// Mitsubishi GX Works2 project: Conv_TF_Connect_Kanban   PLC: FX3U/FX3UC

// global labels: Proce_C1
VAR_GLOBAL
  Add_Plates_C1 : INT;
  Pre_Add_Plates_C1 : INT;
  Add_Box_C1 : INT;
  Out_Product_C1 : INT;
  Codition_C2 : BOOL;
END_VAR

// global labels: Fake_Data
VAR_GLOBAL
  Fake_M45 : TIMER;
END_VAR

PROGRAM ARLAM
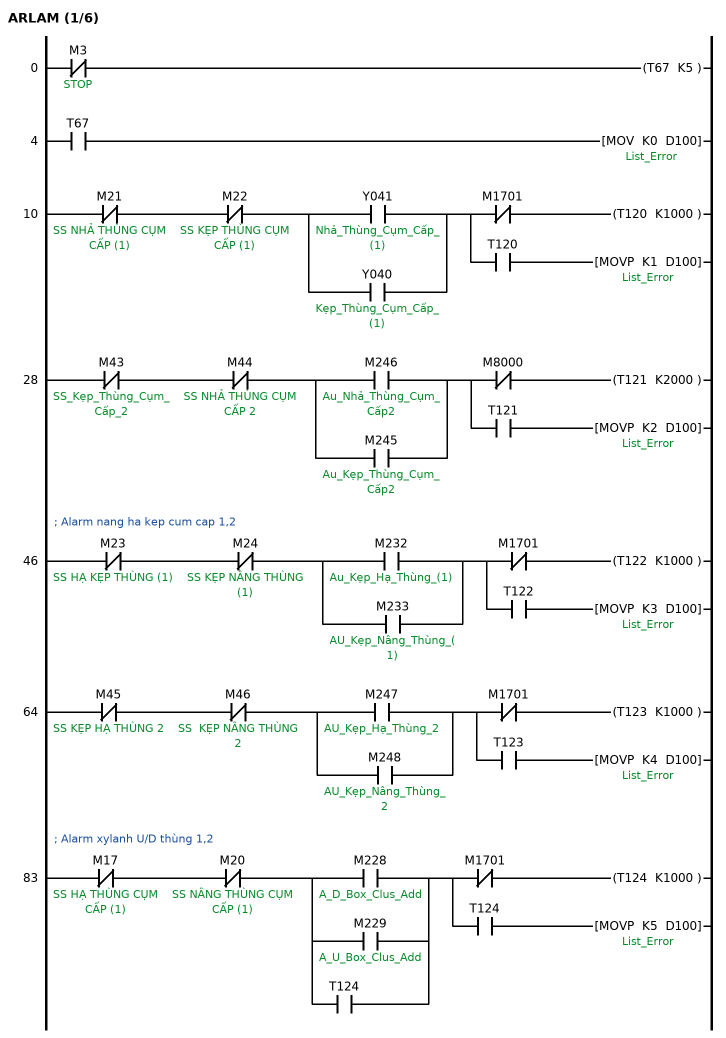
0     LDI     M3  ; STOP
      OUT     T67 K5
4     LD      T67
      MOV     K0 D100  ; List_Error
10    LDI     M21  ; SS NHẢ THÙNG CỤM CẤP (1)
      ANI     M22  ; SS KẸP THÙNG CỤM CẤP (1)
      LD      Y041  ; Nhả_Thùng_Cụm_Cấp_(1)
      OR      Y040  ; Kẹp_Thùng_Cụm_Cấp_(1)
      ANB
      MPS
      ANI     M1701
      OUT     T120 K1000
      MPP
      AND     T120
      MOVP    K1 D100
28    LDI     M43  ; SS_Kẹp_Thùng_Cụm_Cấp_2
      ANI     M44  ; SS NHẢ THÙNG CỤM CẤP 2
      LD      M246  ; Au_Nhả_Thùng_Cụm_Cấp2
      OR      M245  ; Au_Kẹp_Thùng_Cụm_Cấp2
      ANB
      MPS
      ANI     M8000
      OUT     T121 K2000
      MPP
      AND     T121
      MOVP    K2 D100
; Alarm nang ha kep cum cap 1,2
46    LDI     M23  ; SS HẠ KẸP THÙNG (1)
      ANI     M24  ; SS KẸP NÂNG THÙNG (1)
      LD      M232  ; Au_Kẹp_Hạ_Thùng_(1)
      OR      M233  ; AU_Kẹp_Nâng_Thùng_(1)
      ANB
      MPS
      ANI     M1701
      OUT     T122 K1000
      MPP
      AND     T122
      MOVP    K3 D100
64    LDI     M45  ; SS KẸP HẠ THÙNG 2
      ANI     M46  ; SS  KẸP NÂNG THÙNG 2
      LD      M247  ; AU_Kẹp_Hạ_Thùng_2
      OR      M248  ; AU_Kẹp_Nâng_Thùng_2
      ANB
      MPS
      ANI     M1701
      OUT     T123 K1000
      MPP
      AND     T123
      MOVP    K4 D100
; Alarm xylanh U/D thùng 1,2
83    LDI     M17  ; SS HẠ THÙNG CỤM CẤP (1)
      ANI     M20  ; SS NÂNG THÙNG CỤM CẤP (1)
      LD      M228  ; A_D_Box_Clus_Add
      OR      M229  ; A_U_Box_Clus_Add
      OR      T124
      ANB
      MPS
      ANI     M1701
      OUT     T124 K1000
      MPP
      AND     T124
      MOVP    K5 D100
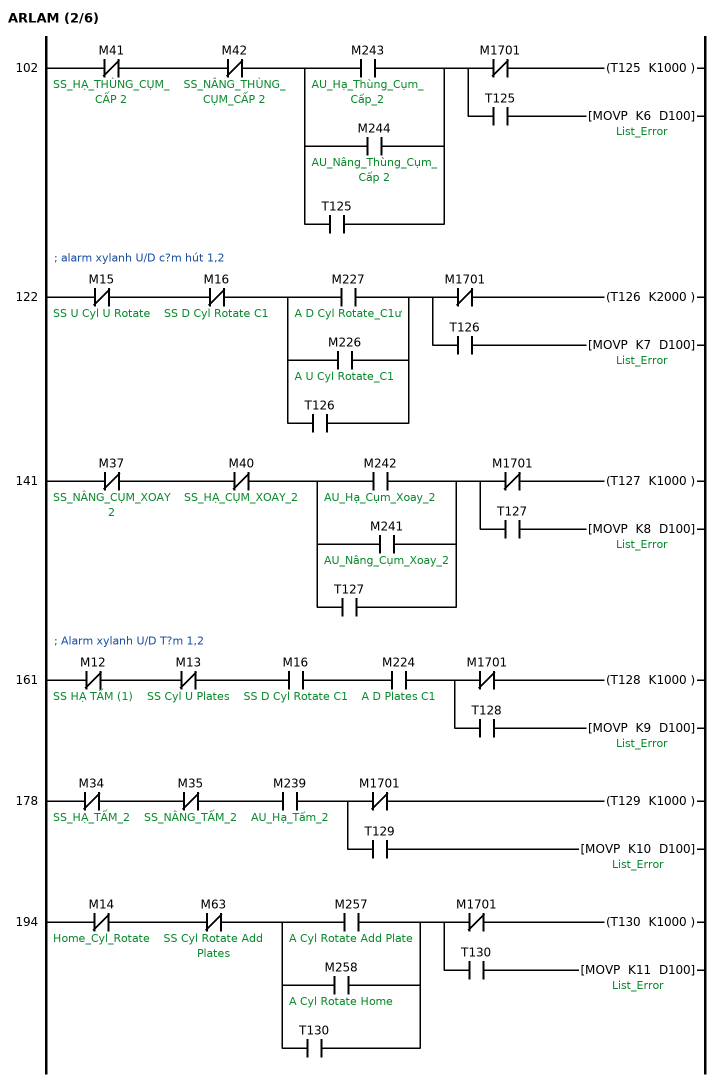
102   LDI     M41  ; SS_HẠ_THÙNG_CỤM_CẤP 2
      ANI     M42  ; SS_NÂNG_THÙNG_CỤM_CẤP 2
      LD      M243  ; AU_Hạ_Thùng_Cụm_Cấp_2
      OR      M244  ; AU_Nâng_Thùng_Cụm_Cấp 2
      OR      T125
      ANB
      MPS
      ANI     M1701
      OUT     T125 K1000
      MPP
      AND     T125
      MOVP    K6 D100
; alarm xylanh U/D c?m hút 1,2
122   LDI     M15  ; SS U Cyl U Rotate
      ANI     M16  ; SS D Cyl Rotate C1
      LD      M227  ; A D Cyl Rotate_C1ư
      OR      M226  ; A U Cyl Rotate_C1
      OR      T126
      ANB
      MPS
      ANI     M1701
      OUT     T126 K2000
      MPP
      AND     T126
      MOVP    K7 D100
141   LDI     M37  ; SS_NÂNG_CỤM_XOAY 2
      ANI     M40  ; SS_HẠ_CỤM_XOAY_2
      LD      M242  ; AU_Hạ_Cụm_Xoay_2
      OR      M241  ; AU_Nâng_Cụm_Xoay_2
      OR      T127
      ANB
      MPS
      ANI     M1701
      OUT     T127 K1000
      MPP
      AND     T127
      MOVP    K8 D100
; Alarm xylanh U/D T?m 1,2
161   LDI     M12  ; SS HẠ TẤM (1)
      ANI     M13  ; SS Cyl U Plates
      AND     M16  ; SS D Cyl Rotate C1
      AND     M224  ; A D Plates C1
      MPS
      ANI     M1701
      OUT     T128 K1000
      MPP
      AND     T128
      MOVP    K9 D100
178   LDI     M34  ; SS_HẠ_TẤM_2
      ANI     M35  ; SS_NÂNG_TẤM_2
      AND     M239  ; AU_Hạ_Tấm_2
      MPS
      ANI     M1701
      OUT     T129 K1000
      MPP
      AND     T129
      MOVP    K10 D100
194   LDI     M14  ; Home_Cyl_Rotate
      ANI     M63  ; SS Cyl Rotate Add Plates
      LD      M257  ; A Cyl Rotate Add Plate
      OR      M258  ; A Cyl Rotate Home
      OR      T130
      ANB
      MPS
      ANI     M1701
      OUT     T130 K1000
      MPP
      AND     T130
      MOVP    K11 D100
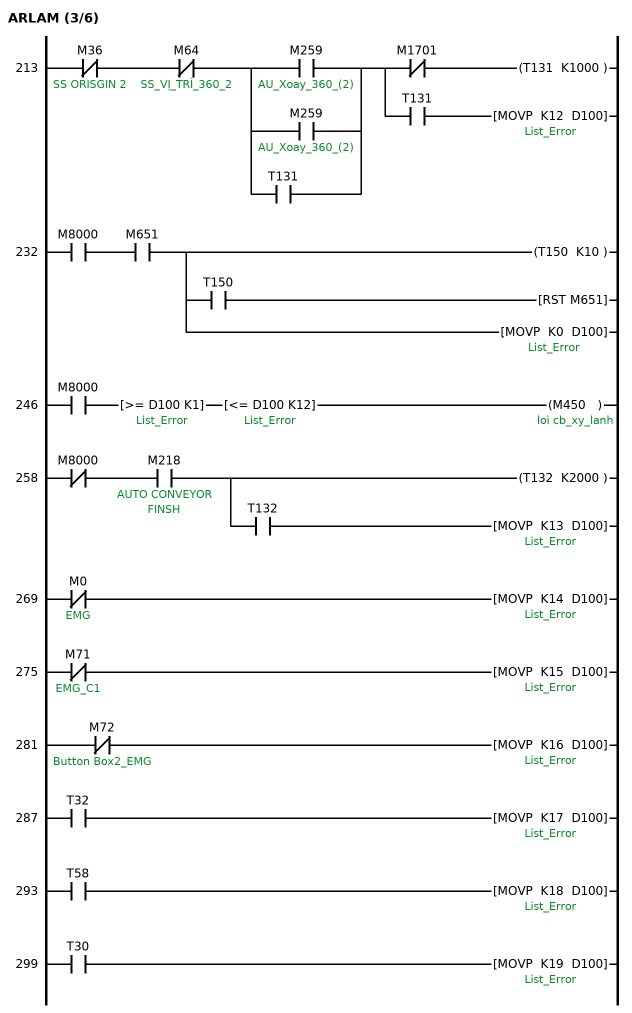
213   LDI     M36  ; SS ORISGIN 2
      ANI     M64  ; SS_VỊ_TRÍ_360_2
      LD      M259  ; AU_Xoay_360_(2)
      OR      M259  ; AU_Xoay_360_(2)
      OR      T131
      ANB
      MPS
      ANI     M1701
      OUT     T131 K1000
      MPP
      AND     T131
      MOVP    K12 D100
232   LD      M8000
      AND     M651
      OUT     T150 K10
      MPS
      AND     T150
      RST     M651
      MPP
      MOVP    K0 D100
246   LD      M8000
      AND>=   D100 K1  ; List_Error
      AND<=   D100 K12  ; List_Error
      OUT     M450  ; loi cb_xy_lanh
258   LDI     M8000
      AND     M218  ; AUTO CONVEYOR FINSH
      OUT     T132 K2000
      AND     T132
      MOVP    K13 D100
269   LDI     M0  ; EMG
      MOVP    K14 D100
275   LDI     M71  ; EMG_C1
      MOVP    K15 D100
281   LDI     M72  ; Button Box2_EMG
      MOVP    K16 D100
287   LD      T32
      MOVP    K17 D100
293   LD      T58
      MOVP    K18 D100
299   LD      T30
      MOVP    K19 D100
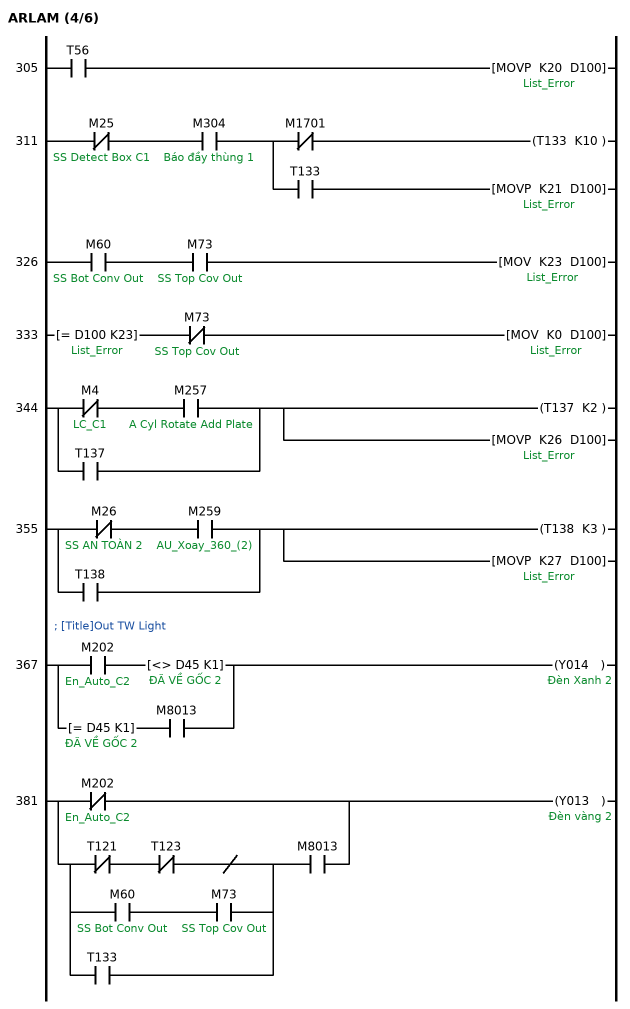
305   LD      T56
      MOVP    K20 D100
311   LDI     M25  ; SS Detect Box C1
      AND     M304  ; Báo đầy thùng 1
      MPS
      ANI     M1701
      OUT     T133 K10
      MPP
      AND     T133
      MOVP    K21 D100
326   LD      M60  ; SS Bot Conv Out
      AND     M73  ; SS Top Cov Out
      MOV     K23 D100
333   LD=     D100 K23  ; List_Error
      ANI     M73  ; SS Top Cov Out
      MOV     K0 D100
344   LDI     M4  ; LC_C1
      AND     M257  ; A Cyl Rotate Add Plate
      OR      T137
      OUT     T137 K2
      MOVP    K26 D100
355   LDI     M26  ; SS AN TOÀN 2
      AND     M259  ; AU_Xoay_360_(2)
      OR      T138
      OUT     T138 K3
      MOVP    K27 D100
; [Title]Out TW Light
367   LD      M202  ; En_Auto_C2
      AND<>   D45 K1  ; ĐÃ VỀ GỐC 2
      LD=     D45 K1  ; ĐÃ VỀ GỐC 2
      AND     M8013
      ORB
      OUT     Y014  ; Đèn Xanh 2
381   LDI     M202  ; En_Auto_C2
      LDI     T121
      ANI     T123
      INV
      LD      M60  ; SS Bot Conv Out
      AND     M73  ; SS Top Cov Out
      ORB
      OR      T133
      AND     M8013
      ORB
      OUT     Y013  ; Đèn vàng 2
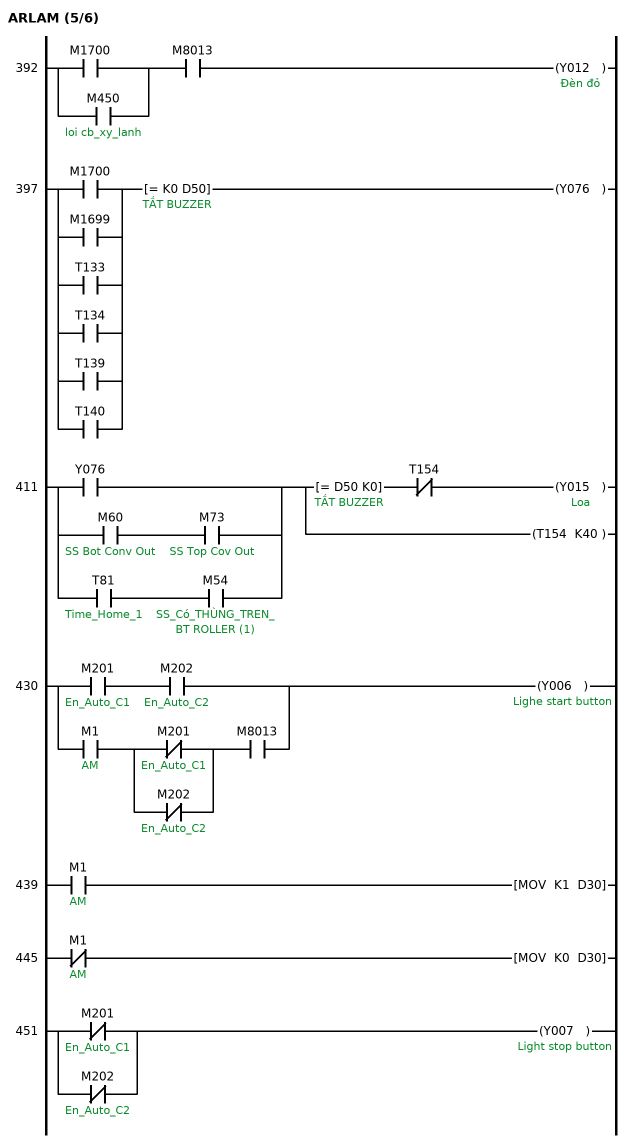
392   LD      M1700
      OR      M450  ; loi cb_xy_lanh
      AND     M8013
      OUT     Y012  ; Đèn đỏ
397   LD      M1700
      OR      M1699
      OR      T133
      OR      T134
      OR      T139
      OR      T140
      AND=    K0 D50  ; TẮT BUZZER
      OUT     Y076
411   LD      Y076
      LD      M60  ; SS Bot Conv Out
      AND     M73  ; SS Top Cov Out
      ORB
      LD      T81  ; Time_Home_1
      AND     M54  ; SS_Có_THÙNG_TREN_BT ROLLER (1)
      ORB
      MPS
      AND=    D50 K0  ; TẮT BUZZER
      ANI     T154
      OUT     Y015  ; Loa
      MPP
      OUT     T154 K40
430   LD      M201  ; En_Auto_C1
      AND     M202  ; En_Auto_C2
      LD      M1  ; AM
      LDI     M201  ; En_Auto_C1
      ORI     M202  ; En_Auto_C2
      ANB
      AND     M8013
      ORB
      OUT     Y006  ; Lighe start button
439   LD      M1  ; AM
      MOV     K1 D30
445   LDI     M1  ; AM
      MOV     K0 D30
451   LDI     M201  ; En_Auto_C1
      ORI     M202  ; En_Auto_C2
      OUT     Y007  ; Light stop button
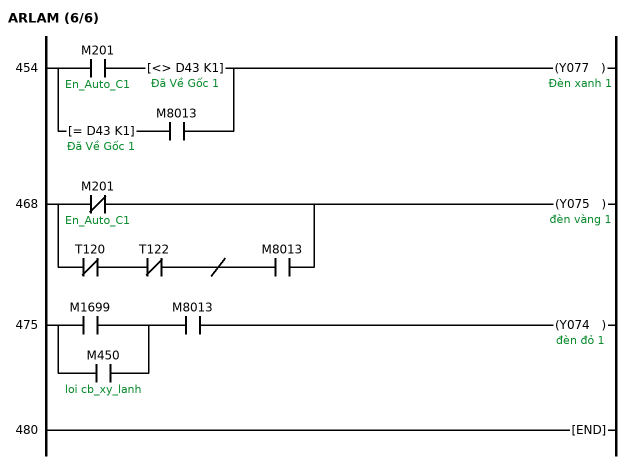
454   LD      M201  ; En_Auto_C1
      AND<>   D43 K1  ; Đã Về Gốc 1
      LD=     D43 K1  ; Đã Về Gốc 1
      AND     M8013
      ORB
      OUT     Y077  ; Đèn xanh 1
468   LDI     M201  ; En_Auto_C1
      LDI     T120
      ANI     T122
      INV
      AND     M8013
      ORB
      OUT     Y075  ; đèn vàng 1
475   LD      M1699
      OR      M450  ; loi cb_xy_lanh
      AND     M8013
      OUT     Y074  ; đèn đỏ 1
480   END
END_PROGRAM

PROGRAM AUTO
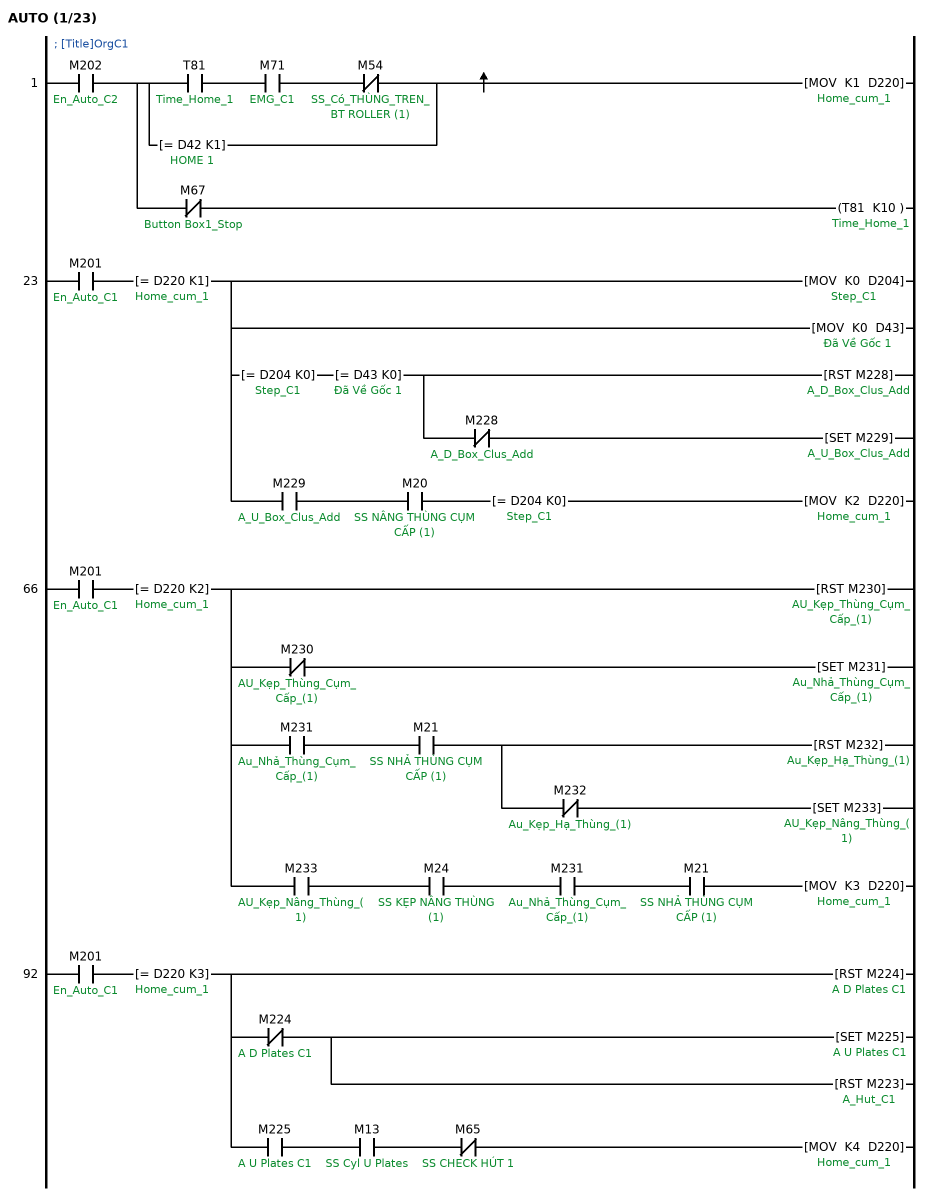
; [Title]OrgC1
1     LD      M202  ; En_Auto_C2
      MPS
      LD      T81  ; Time_Home_1
      AND     M71  ; EMG_C1
      ANI     M54  ; SS_Có_THÙNG_TREN_BT ROLLER (1)
      OR=     D42 K1  ; HOME 1
      ANB
      MEP
      MOV     K1 D220  ; Home_cum_1
      MPP
      ANI     M67  ; Button Box1_Stop
      OUT     T81 K10  ; Time_Home_1
23    LD      M201  ; En_Auto_C1
      AND=    D220 K1  ; Home_cum_1
      MOV     K0 D204  ; Step_C1
      MOV     K0 D43  ; Đã Về Gốc 1
      MPS
      AND=    D204 K0  ; Step_C1
      AND=    D43 K0  ; Đã Về Gốc 1
      RST     M228  ; A_D_Box_Clus_Add
      ANI     M228  ; A_D_Box_Clus_Add
      SET     M229  ; A_U_Box_Clus_Add
      MPP
      AND     M229  ; A_U_Box_Clus_Add
      AND     M20  ; SS NÂNG THÙNG CỤM CẤP (1)
      AND=    D204 K0  ; Step_C1
      MOV     K2 D220
66    LD      M201  ; En_Auto_C1
      AND=    D220 K2  ; Home_cum_1
      RST     M230  ; AU_Kẹp_Thùng_Cụm_Cấp_(1)
      MPS
      ANI     M230  ; AU_Kẹp_Thùng_Cụm_Cấp_(1)
      SET     M231  ; Au_Nhả_Thùng_Cụm_Cấp_(1)
      MRD
      AND     M231  ; Au_Nhả_Thùng_Cụm_Cấp_(1)
      AND     M21  ; SS NHẢ THÙNG CỤM CẤP (1)
      RST     M232  ; Au_Kẹp_Hạ_Thùng_(1)
      ANI     M232  ; Au_Kẹp_Hạ_Thùng_(1)
      SET     M233  ; AU_Kẹp_Nâng_Thùng_(1)
      MPP
      AND     M233  ; AU_Kẹp_Nâng_Thùng_(1)
      AND     M24  ; SS KẸP NÂNG THÙNG (1)
      AND     M231  ; Au_Nhả_Thùng_Cụm_Cấp_(1)
      AND     M21  ; SS NHẢ THÙNG CỤM CẤP (1)
      MOV     K3 D220
92    LD      M201  ; En_Auto_C1
      AND=    D220 K3  ; Home_cum_1
      RST     M224  ; A D Plates C1
      MPS
      ANI     M224  ; A D Plates C1
      SET     M225  ; A U Plates C1
      RST     M223  ; A_Hut_C1
      MPP
      AND     M225  ; A U Plates C1
      AND     M13  ; SS Cyl U Plates
      ANI     M65  ; SS CHECK HÚT 1
      MOV     K4 D220
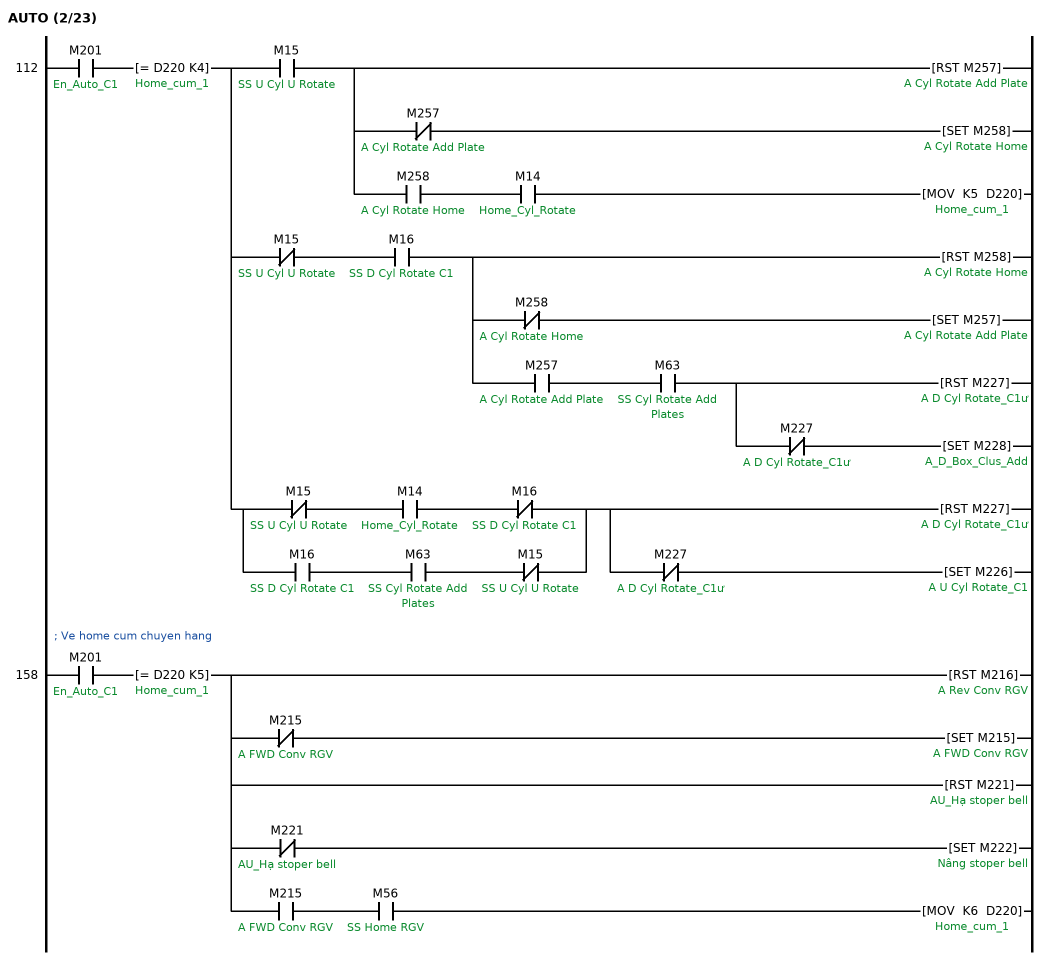
112   LD      M201  ; En_Auto_C1
      AND=    D220 K4  ; Home_cum_1
      MPS
      AND     M15  ; SS U Cyl U Rotate
      RST     M257  ; A Cyl Rotate Add Plate
      MPS
      ANI     M257  ; A Cyl Rotate Add Plate
      SET     M258  ; A Cyl Rotate Home
      MPP
      AND     M258  ; A Cyl Rotate Home
      AND     M14  ; Home_Cyl_Rotate
      MOV     K5 D220
      MRD
      ANI     M15  ; SS U Cyl U Rotate
      AND     M16  ; SS D Cyl Rotate C1
      RST     M258  ; A Cyl Rotate Home
      MPS
      ANI     M258  ; A Cyl Rotate Home
      SET     M257  ; A Cyl Rotate Add Plate
      MPP
      AND     M257  ; A Cyl Rotate Add Plate
      AND     M63  ; SS Cyl Rotate Add Plates
      RST     M227  ; A D Cyl Rotate_C1ư
      ANI     M227  ; A D Cyl Rotate_C1ư
      SET     M228  ; A_D_Box_Clus_Add
      MPP
      LDI     M15  ; SS U Cyl U Rotate
      AND     M14  ; Home_Cyl_Rotate
      ANI     M16  ; SS D Cyl Rotate C1
      LD      M16  ; SS D Cyl Rotate C1
      AND     M63  ; SS Cyl Rotate Add Plates
      ANI     M15  ; SS U Cyl U Rotate
      ORB
      ANB
      RST     M227  ; A D Cyl Rotate_C1ư
      ANI     M227  ; A D Cyl Rotate_C1ư
      SET     M226  ; A U Cyl Rotate_C1
; Ve home cum chuyen hang
158   LD      M201  ; En_Auto_C1
      AND=    D220 K5  ; Home_cum_1
      RST     M216  ; A Rev Conv RGV
      MPS
      ANI     M215  ; A FWD Conv RGV
      SET     M215  ; A FWD Conv RGV
      MPP
      RST     M221  ; AU_Hạ stoper bell
      MPS
      ANI     M221  ; AU_Hạ stoper bell
      SET     M222  ; Nâng stoper bell
      MPP
      AND     M215  ; A FWD Conv RGV
      AND     M56  ; SS Home RGV
      MOV     K6 D220
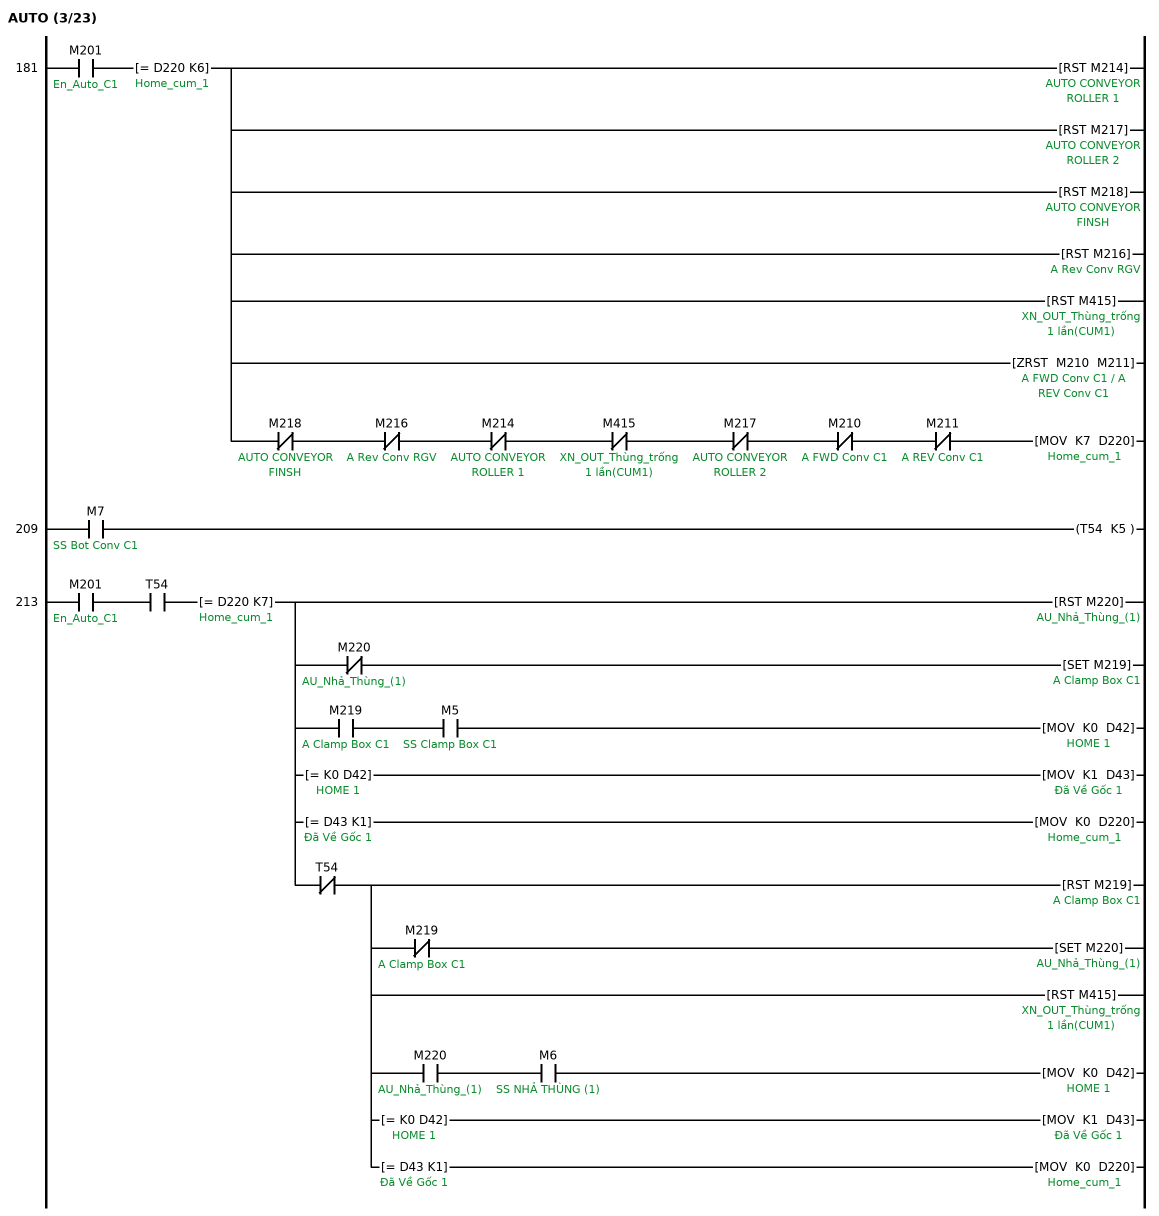
181   LD      M201  ; En_Auto_C1
      AND=    D220 K6  ; Home_cum_1
      RST     M214  ; AUTO CONVEYOR ROLLER 1
      RST     M217  ; AUTO CONVEYOR ROLLER 2
      RST     M218  ; AUTO CONVEYOR FINSH
      RST     M216  ; A Rev Conv RGV
      RST     M415  ; XN_OUT_Thùng_trống 1 lần(CUM1)
      ZRST    M210 M211  ; A FWD Conv C1 / A REV Conv C1
      ANI     M218  ; AUTO CONVEYOR FINSH
      ANI     M216  ; A Rev Conv RGV
      ANI     M214  ; AUTO CONVEYOR ROLLER 1
      ANI     M415  ; XN_OUT_Thùng_trống 1 lần(CUM1)
      ANI     M217  ; AUTO CONVEYOR ROLLER 2
      ANI     M210  ; A FWD Conv C1
      ANI     M211  ; A REV Conv C1
      MOV     K7 D220
209   LD      M7  ; SS Bot Conv C1
      OUT     T54 K5
213   LD      M201  ; En_Auto_C1
      AND     T54
      AND=    D220 K7  ; Home_cum_1
      RST     M220  ; AU_Nhả_Thùng_(1)
      MPS
      ANI     M220  ; AU_Nhả_Thùng_(1)
      SET     M219  ; A Clamp Box C1
      MRD
      AND     M219  ; A Clamp Box C1
      AND     M5  ; SS Clamp Box C1
      MOV     K0 D42
      MRD
      AND=    K0 D42  ; HOME 1
      MOV     K1 D43
      MRD
      AND=    D43 K1  ; Đã Về Gốc 1
      MOV     K0 D220
      MPP
      ANI     T54
      RST     M219  ; A Clamp Box C1
      MPS
      ANI     M219  ; A Clamp Box C1
      SET     M220  ; AU_Nhả_Thùng_(1)
      MPP
      RST     M415  ; XN_OUT_Thùng_trống 1 lần(CUM1)
      MPS
      AND     M220  ; AU_Nhả_Thùng_(1)
      AND     M6  ; SS NHẢ THÙNG (1)
      MOV     K0 D42
      MRD
      AND=    K0 D42  ; HOME 1
      MOV     K1 D43
      MPP
      AND=    D43 K1  ; Đã Về Gốc 1
      MOV     K0 D220
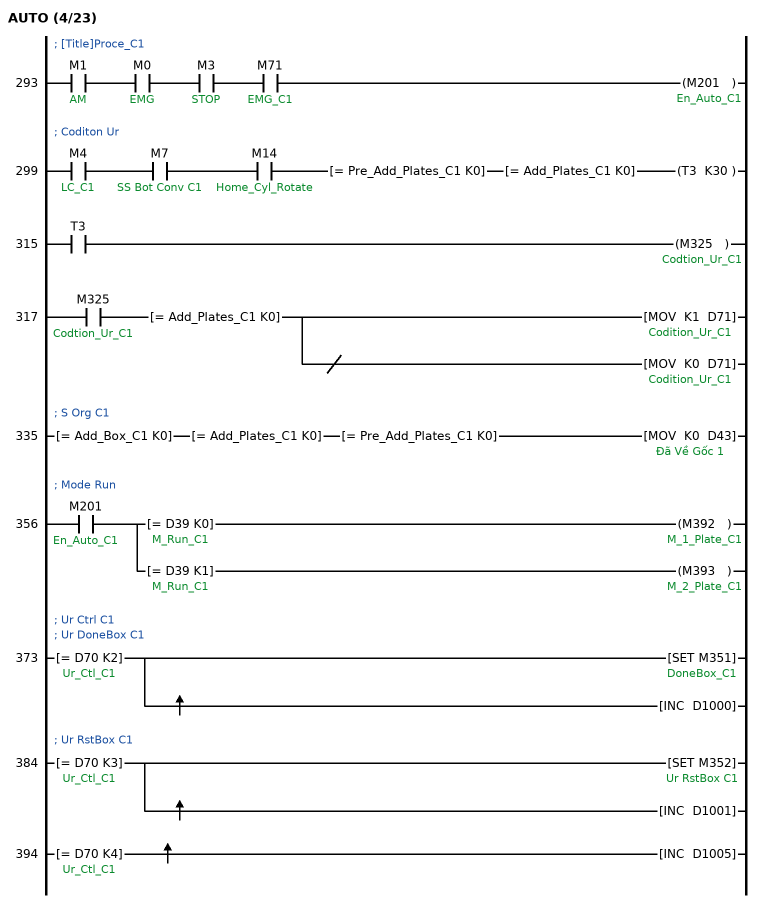
; [Title]Proce_C1
293   LD      M1  ; AM
      AND     M0  ; EMG
      AND     M3  ; STOP
      AND     M71  ; EMG_C1
      OUT     M201  ; En_Auto_C1
; Coditon Ur
299   LD      M4  ; LC_C1
      AND     M7  ; SS Bot Conv C1
      AND     M14  ; Home_Cyl_Rotate
      AND=    Pre_Add_Plates_C1 K0
      AND=    Add_Plates_C1 K0
      OUT     T3 K30
315   LD      T3
      OUT     M325  ; Codtion_Ur_C1
317   LD      M325  ; Codtion_Ur_C1
      AND=    Add_Plates_C1 K0
      MOV     K1 D71  ; Codition_Ur_C1
      INV
      MOV     K0 D71
; S Org C1
335   LD=     Add_Box_C1 K0
      AND=    Add_Plates_C1 K0
      AND=    Pre_Add_Plates_C1 K0
      MOV     K0 D43
; Mode Run
356   LD      M201  ; En_Auto_C1
      MPS
      AND=    D39 K0  ; M_Run_C1
      OUT     M392  ; M_1_Plate_C1
      MPP
      AND=    D39 K1  ; M_Run_C1
      OUT     M393  ; M_2_Plate_C1
; Ur Ctrl C1
; Ur DoneBox C1
373   LD=     D70 K2  ; Ur_Ctl_C1
      SET     M351  ; DoneBox_C1
      MEP
      INC     D1000
; Ur RstBox C1
384   LD=     D70 K3  ; Ur_Ctl_C1
      SET     M352  ; Ur RstBox C1
      MEP
      INC     D1001
394   LD=     D70 K4  ; Ur_Ctl_C1
      MEP
      INC     D1005
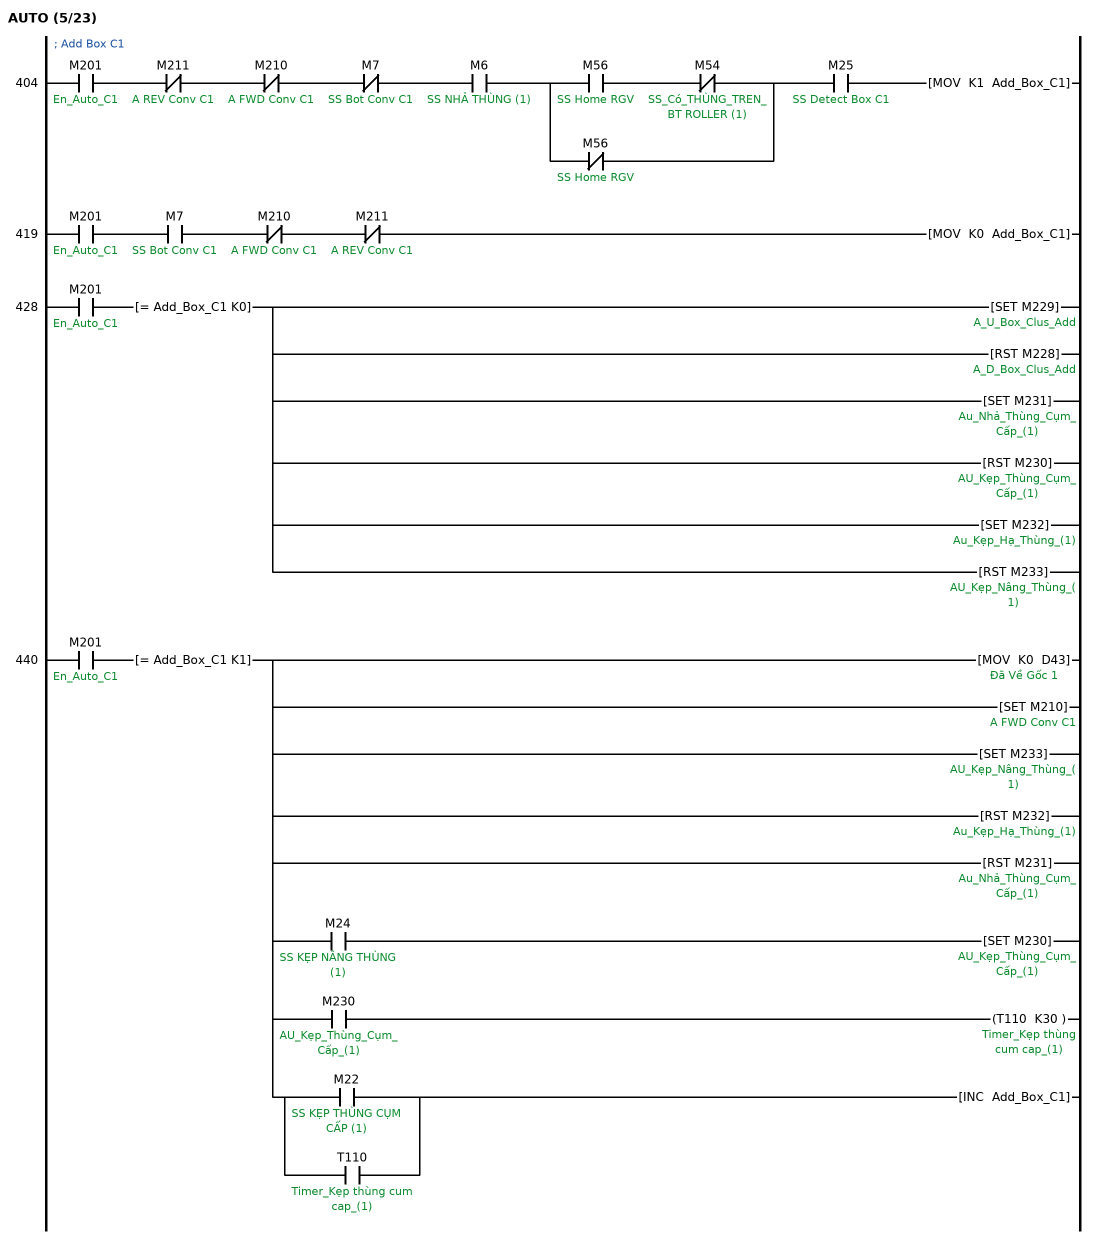
; Add Box C1
404   LD      M201  ; En_Auto_C1
      ANI     M211  ; A REV Conv C1
      ANI     M210  ; A FWD Conv C1
      ANI     M7  ; SS Bot Conv C1
      AND     M6  ; SS NHẢ THÙNG (1)
      LD      M56  ; SS Home RGV
      ANI     M54  ; SS_Có_THÙNG_TREN_BT ROLLER (1)
      ORI     M56  ; SS Home RGV
      ANB
      AND     M25  ; SS Detect Box C1
      MOV     K1 Add_Box_C1
419   LD      M201  ; En_Auto_C1
      AND     M7  ; SS Bot Conv C1
      ANI     M210  ; A FWD Conv C1
      ANI     M211  ; A REV Conv C1
      MOV     K0 Add_Box_C1
428   LD      M201  ; En_Auto_C1
      AND=    Add_Box_C1 K0
      SET     M229  ; A_U_Box_Clus_Add
      RST     M228  ; A_D_Box_Clus_Add
      SET     M231  ; Au_Nhả_Thùng_Cụm_Cấp_(1)
      RST     M230  ; AU_Kẹp_Thùng_Cụm_Cấp_(1)
      SET     M232  ; Au_Kẹp_Hạ_Thùng_(1)
      RST     M233  ; AU_Kẹp_Nâng_Thùng_(1)
440   LD      M201  ; En_Auto_C1
      AND=    Add_Box_C1 K1
      MOV     K0 D43
      SET     M210  ; A FWD Conv C1
      SET     M233  ; AU_Kẹp_Nâng_Thùng_(1)
      RST     M232  ; Au_Kẹp_Hạ_Thùng_(1)
      RST     M231  ; Au_Nhả_Thùng_Cụm_Cấp_(1)
      MPS
      AND     M24  ; SS KẸP NÂNG THÙNG (1)
      SET     M230  ; AU_Kẹp_Thùng_Cụm_Cấp_(1)
      MRD
      AND     M230  ; AU_Kẹp_Thùng_Cụm_Cấp_(1)
      OUT     T110 K30  ; Timer_Kẹp thùng cum cap_(1)
      MPP
      LD      M22  ; SS KẸP THÙNG CỤM CẤP (1)
      OR      T110  ; Timer_Kẹp thùng cum cap_(1)
      ANB
      INC     Add_Box_C1
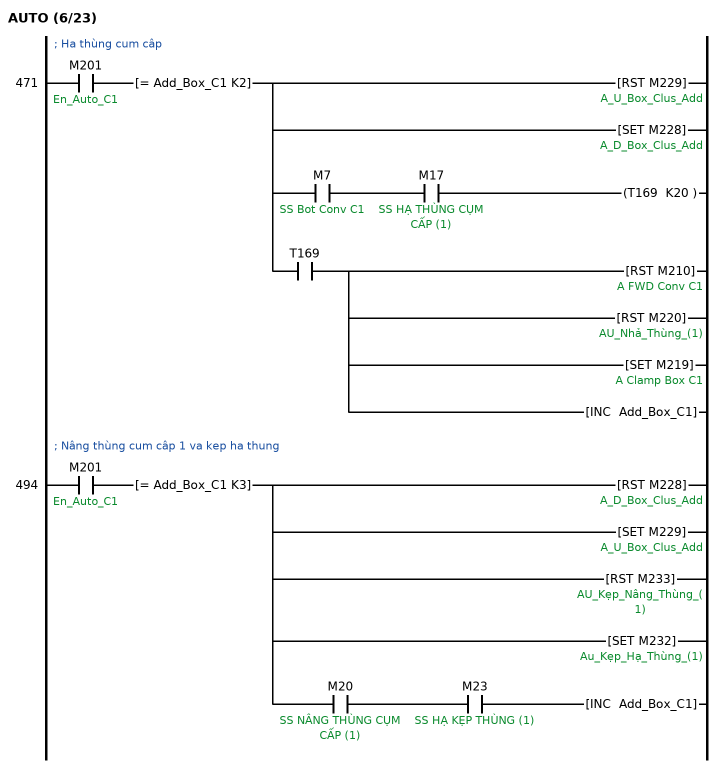
; Ha thùng cum câp
471   LD      M201  ; En_Auto_C1
      AND=    Add_Box_C1 K2
      RST     M229  ; A_U_Box_Clus_Add
      SET     M228  ; A_D_Box_Clus_Add
      MPS
      AND     M7  ; SS Bot Conv C1
      AND     M17  ; SS HẠ THÙNG CỤM CẤP (1)
      OUT     T169 K20
      MPP
      AND     T169
      RST     M210  ; A FWD Conv C1
      RST     M220  ; AU_Nhả_Thùng_(1)
      SET     M219  ; A Clamp Box C1
      INC     Add_Box_C1
; Nâng thùng cum câp 1 va kep ha thung
494   LD      M201  ; En_Auto_C1
      AND=    Add_Box_C1 K3
      RST     M228  ; A_D_Box_Clus_Add
      SET     M229  ; A_U_Box_Clus_Add
      RST     M233  ; AU_Kẹp_Nâng_Thùng_(1)
      SET     M232  ; Au_Kẹp_Hạ_Thùng_(1)
      AND     M20  ; SS NÂNG THÙNG CỤM CẤP (1)
      AND     M23  ; SS HẠ KẸP THÙNG (1)
      INC     Add_Box_C1
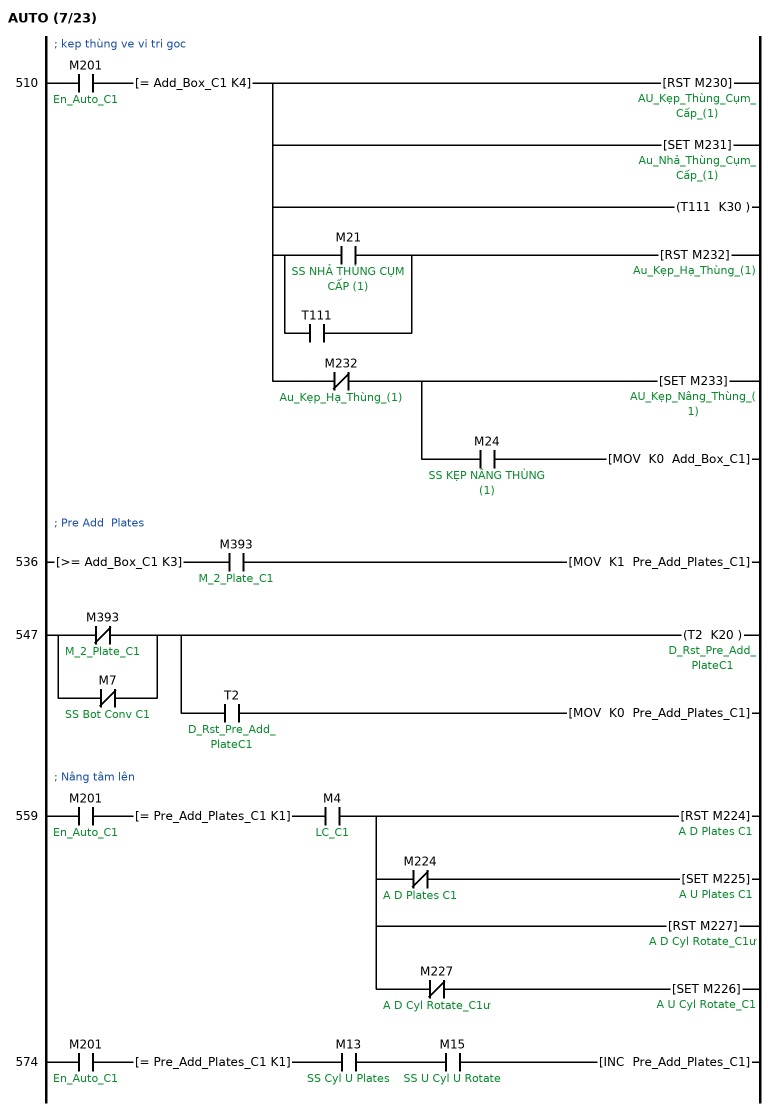
; kep thùng ve vi tri goc
510   LD      M201  ; En_Auto_C1
      AND=    Add_Box_C1 K4
      RST     M230  ; AU_Kẹp_Thùng_Cụm_Cấp_(1)
      SET     M231  ; Au_Nhả_Thùng_Cụm_Cấp_(1)
      OUT     T111 K30
      MPS
      LD      M21  ; SS NHẢ THÙNG CỤM CẤP (1)
      OR      T111
      ANB
      RST     M232  ; Au_Kẹp_Hạ_Thùng_(1)
      MPP
      ANI     M232  ; Au_Kẹp_Hạ_Thùng_(1)
      SET     M233  ; AU_Kẹp_Nâng_Thùng_(1)
      AND     M24  ; SS KẸP NÂNG THÙNG (1)
      MOV     K0 Add_Box_C1
; Pre Add  Plates
536   LD>=    Add_Box_C1 K3
      AND     M393  ; M_2_Plate_C1
      MOV     K1 Pre_Add_Plates_C1
547   LDI     M393  ; M_2_Plate_C1
      ORI     M7  ; SS Bot Conv C1
      OUT     T2 K20  ; D_Rst_Pre_Add_PlateC1
      AND     T2  ; D_Rst_Pre_Add_PlateC1
      MOV     K0 Pre_Add_Plates_C1
; Nâng tâm lên
559   LD      M201  ; En_Auto_C1
      AND=    Pre_Add_Plates_C1 K1
      AND     M4  ; LC_C1
      RST     M224  ; A D Plates C1
      MPS
      ANI     M224  ; A D Plates C1
      SET     M225  ; A U Plates C1
      MPP
      RST     M227  ; A D Cyl Rotate_C1ư
      ANI     M227  ; A D Cyl Rotate_C1ư
      SET     M226  ; A U Cyl Rotate_C1
574   LD      M201  ; En_Auto_C1
      AND=    Pre_Add_Plates_C1 K1
      AND     M13  ; SS Cyl U Plates
      AND     M15  ; SS U Cyl U Rotate
      INC     Pre_Add_Plates_C1
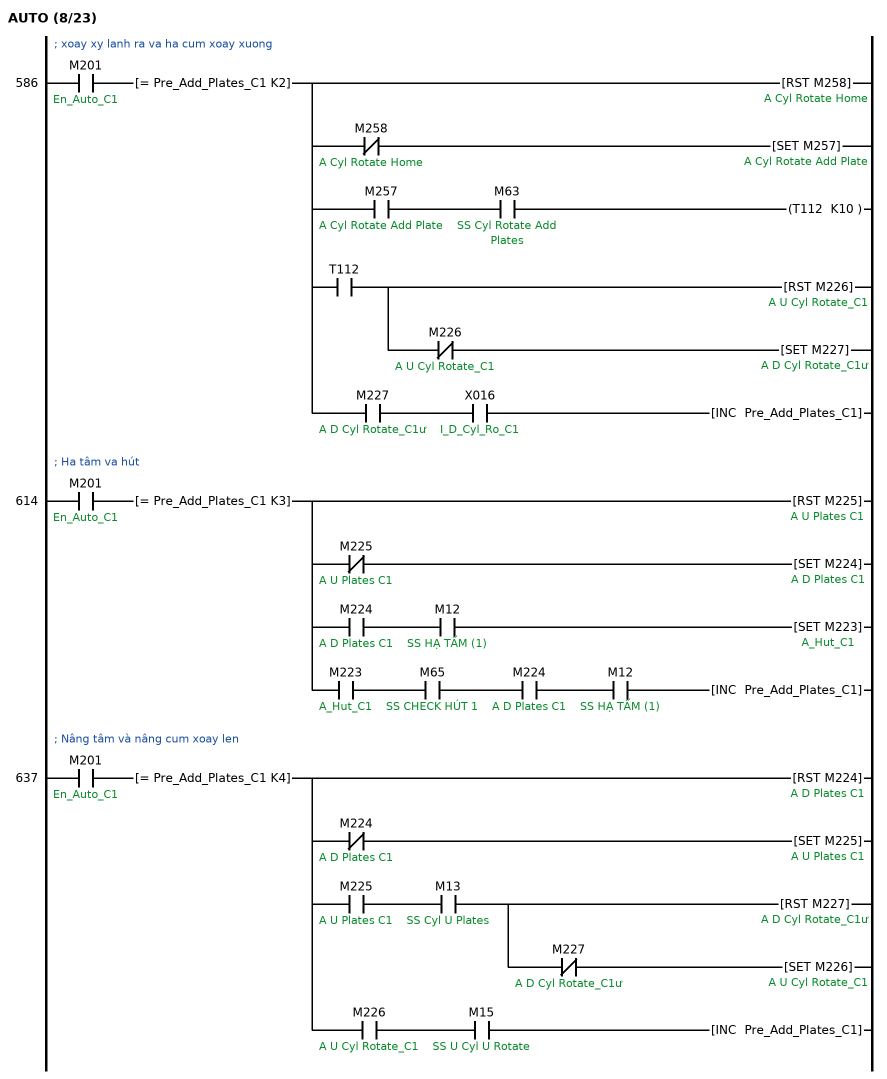
; xoay xy lanh ra va ha cum xoay xuong
586   LD      M201  ; En_Auto_C1
      AND=    Pre_Add_Plates_C1 K2
      RST     M258  ; A Cyl Rotate Home
      MPS
      ANI     M258  ; A Cyl Rotate Home
      SET     M257  ; A Cyl Rotate Add Plate
      MRD
      AND     M257  ; A Cyl Rotate Add Plate
      AND     M63  ; SS Cyl Rotate Add Plates
      OUT     T112 K10
      MRD
      AND     T112
      RST     M226  ; A U Cyl Rotate_C1
      ANI     M226  ; A U Cyl Rotate_C1
      SET     M227  ; A D Cyl Rotate_C1ư
      MPP
      AND     M227  ; A D Cyl Rotate_C1ư
      AND     X016  ; I_D_Cyl_Ro_C1
      INC     Pre_Add_Plates_C1
; Ha tâm va hút
614   LD      M201  ; En_Auto_C1
      AND=    Pre_Add_Plates_C1 K3
      RST     M225  ; A U Plates C1
      MPS
      ANI     M225  ; A U Plates C1
      SET     M224  ; A D Plates C1
      MRD
      AND     M224  ; A D Plates C1
      AND     M12  ; SS HẠ TẤM (1)
      SET     M223  ; A_Hut_C1
      MPP
      AND     M223  ; A_Hut_C1
      AND     M65  ; SS CHECK HÚT 1
      AND     M224  ; A D Plates C1
      AND     M12  ; SS HẠ TẤM (1)
      INC     Pre_Add_Plates_C1
; Nâng tâm và nâng cum xoay len
637   LD      M201  ; En_Auto_C1
      AND=    Pre_Add_Plates_C1 K4
      RST     M224  ; A D Plates C1
      MPS
      ANI     M224  ; A D Plates C1
      SET     M225  ; A U Plates C1
      MRD
      AND     M225  ; A U Plates C1
      AND     M13  ; SS Cyl U Plates
      RST     M227  ; A D Cyl Rotate_C1ư
      ANI     M227  ; A D Cyl Rotate_C1ư
      SET     M226  ; A U Cyl Rotate_C1
      MPP
      AND     M226  ; A U Cyl Rotate_C1
      AND     M15  ; SS U Cyl U Rotate
      INC     Pre_Add_Plates_C1
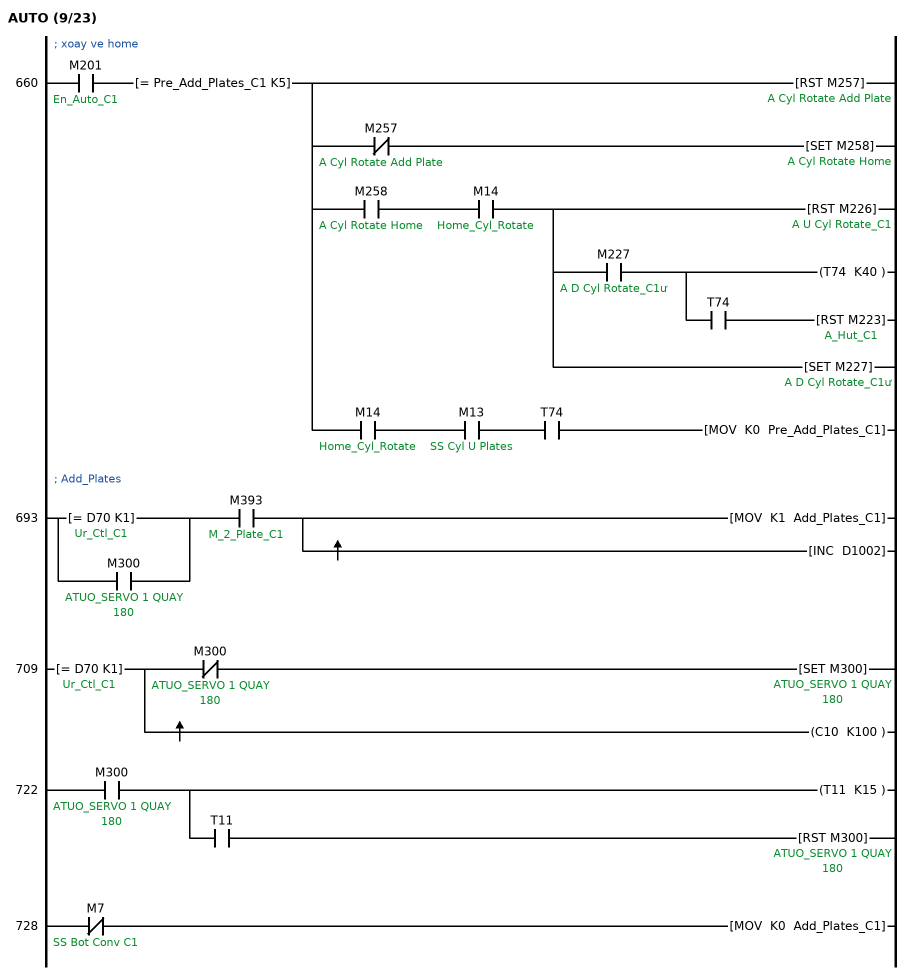
; xoay ve home
660   LD      M201  ; En_Auto_C1
      AND=    Pre_Add_Plates_C1 K5
      RST     M257  ; A Cyl Rotate Add Plate
      MPS
      ANI     M257  ; A Cyl Rotate Add Plate
      SET     M258  ; A Cyl Rotate Home
      MRD
      AND     M258  ; A Cyl Rotate Home
      AND     M14  ; Home_Cyl_Rotate
      RST     M226  ; A U Cyl Rotate_C1
      MPS
      AND     M227  ; A D Cyl Rotate_C1ư
      OUT     T74 K40
      AND     T74
      RST     M223  ; A_Hut_C1
      MPP
      SET     M227  ; A D Cyl Rotate_C1ư
      MPP
      AND     M14  ; Home_Cyl_Rotate
      AND     M13  ; SS Cyl U Plates
      AND     T74
      MOV     K0 Pre_Add_Plates_C1
; Add_Plates
693   LD=     D70 K1  ; Ur_Ctl_C1
      OR      M300  ; ATUO_SERVO 1 QUAY 180
      AND     M393  ; M_2_Plate_C1
      MOV     K1 Add_Plates_C1
      MEP
      INC     D1002
709   LD=     D70 K1  ; Ur_Ctl_C1
      MPS
      ANI     M300  ; ATUO_SERVO 1 QUAY 180
      SET     M300  ; ATUO_SERVO 1 QUAY 180
      MPP
      MEP
      OUT     C10 K100
722   LD      M300  ; ATUO_SERVO 1 QUAY 180
      OUT     T11 K15
      AND     T11
      RST     M300  ; ATUO_SERVO 1 QUAY 180
728   LDI     M7  ; SS Bot Conv C1
      MOV     K0 Add_Plates_C1
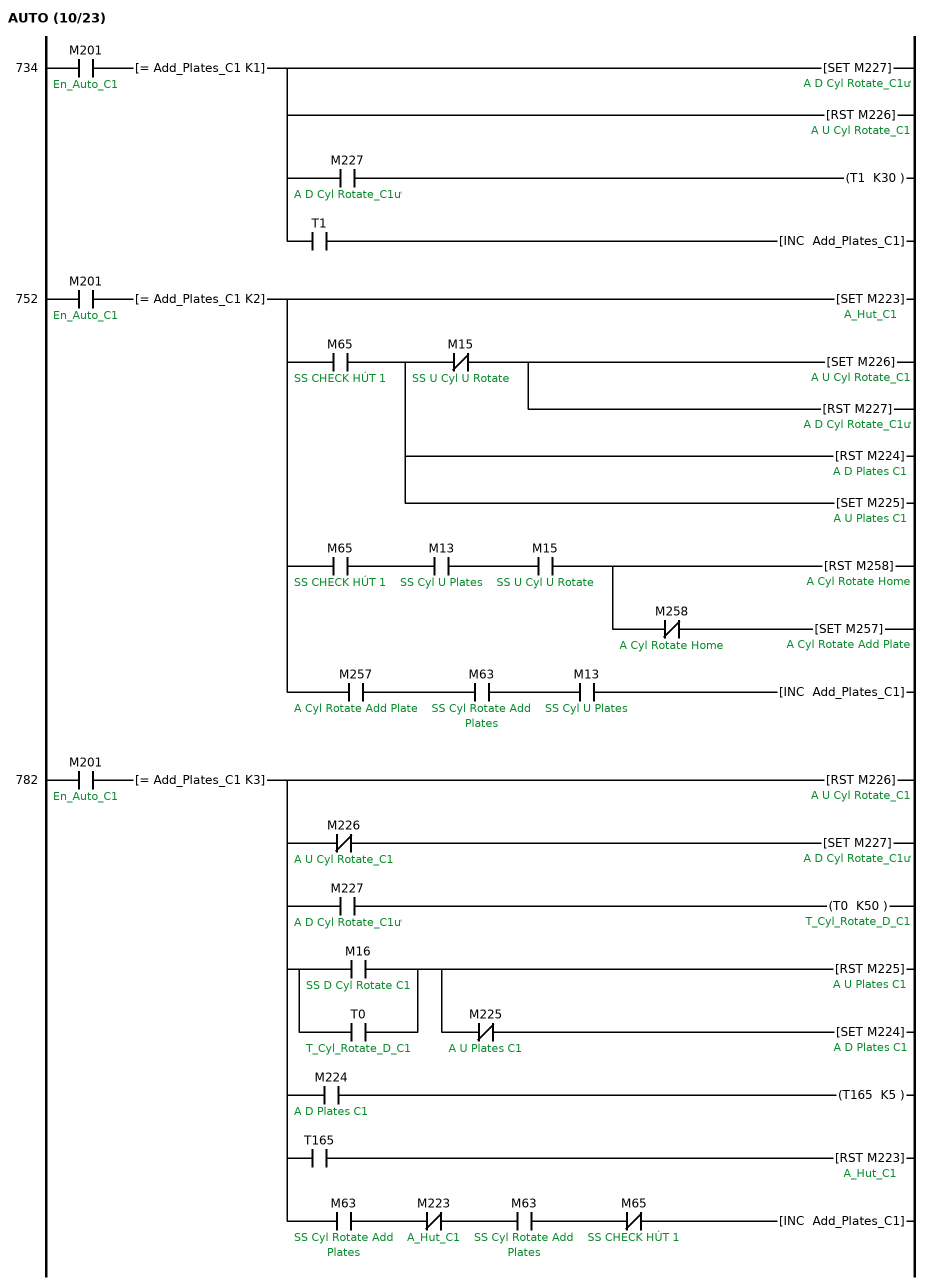
734   LD      M201  ; En_Auto_C1
      AND=    Add_Plates_C1 K1
      SET     M227  ; A D Cyl Rotate_C1ư
      RST     M226  ; A U Cyl Rotate_C1
      MPS
      AND     M227  ; A D Cyl Rotate_C1ư
      OUT     T1 K30
      MPP
      AND     T1
      INC     Add_Plates_C1
752   LD      M201  ; En_Auto_C1
      AND=    Add_Plates_C1 K2
      SET     M223  ; A_Hut_C1
      MPS
      AND     M65  ; SS CHECK HÚT 1
      MPS
      ANI     M15  ; SS U Cyl U Rotate
      SET     M226  ; A U Cyl Rotate_C1
      RST     M227  ; A D Cyl Rotate_C1ư
      MPP
      RST     M224  ; A D Plates C1
      SET     M225  ; A U Plates C1
      MRD
      AND     M65  ; SS CHECK HÚT 1
      AND     M13  ; SS Cyl U Plates
      AND     M15  ; SS U Cyl U Rotate
      RST     M258  ; A Cyl Rotate Home
      ANI     M258  ; A Cyl Rotate Home
      SET     M257  ; A Cyl Rotate Add Plate
      MPP
      AND     M257  ; A Cyl Rotate Add Plate
      AND     M63  ; SS Cyl Rotate Add Plates
      AND     M13  ; SS Cyl U Plates
      INC     Add_Plates_C1
782   LD      M201  ; En_Auto_C1
      AND=    Add_Plates_C1 K3
      RST     M226  ; A U Cyl Rotate_C1
      MPS
      ANI     M226  ; A U Cyl Rotate_C1
      SET     M227  ; A D Cyl Rotate_C1ư
      MRD
      AND     M227  ; A D Cyl Rotate_C1ư
      OUT     T0 K50  ; T_Cyl_Rotate_D_C1
      MRD
      LD      M16  ; SS D Cyl Rotate C1
      OR      T0  ; T_Cyl_Rotate_D_C1
      ANB
      RST     M225  ; A U Plates C1
      ANI     M225  ; A U Plates C1
      SET     M224  ; A D Plates C1
      MRD
      AND     M224  ; A D Plates C1
      OUT     T165 K5
      MRD
      AND     T165
      RST     M223  ; A_Hut_C1
      MPP
      AND     M63  ; SS Cyl Rotate Add Plates
      ANI     M223  ; A_Hut_C1
      AND     M63  ; SS Cyl Rotate Add Plates
      ANI     M65  ; SS CHECK HÚT 1
      INC     Add_Plates_C1
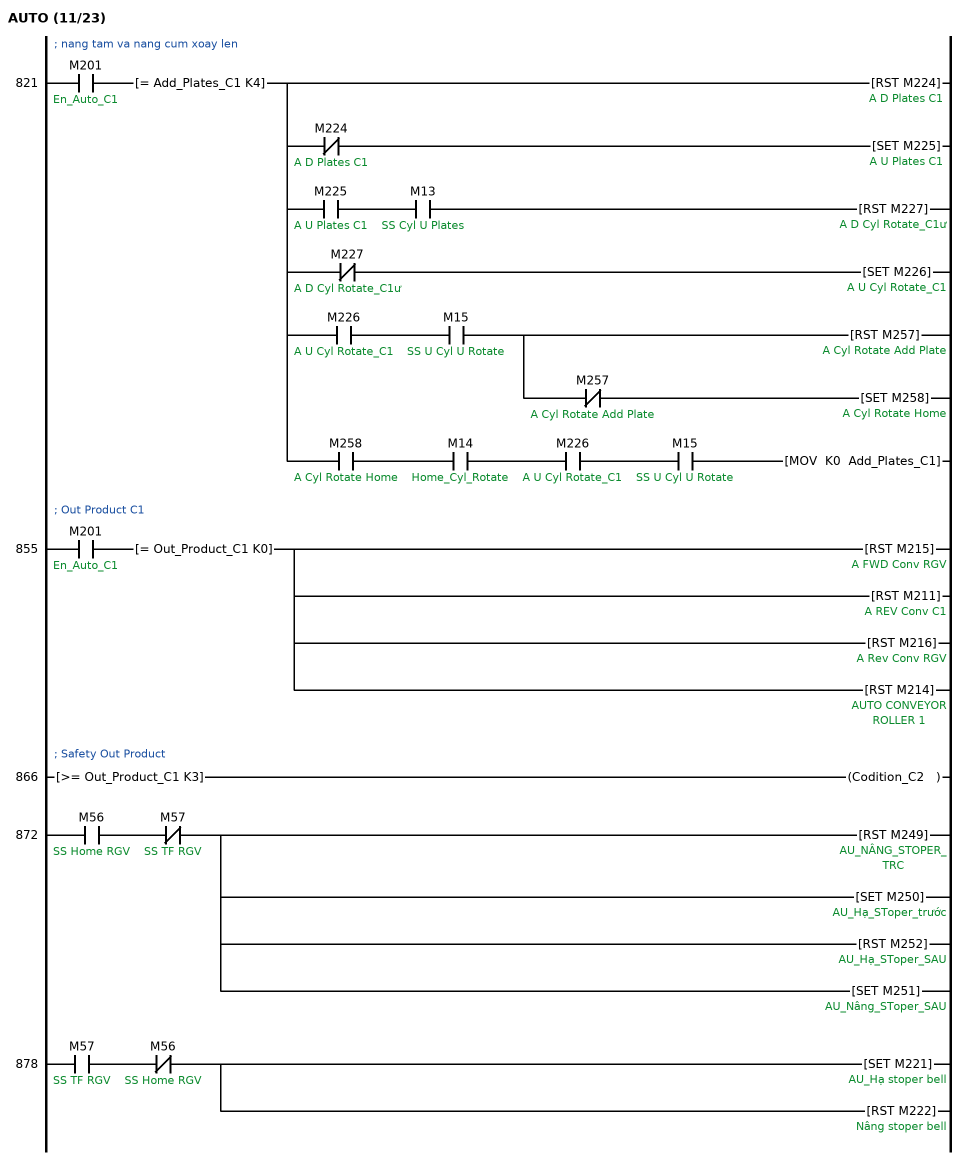
; nang tam va nang cum xoay len
821   LD      M201  ; En_Auto_C1
      AND=    Add_Plates_C1 K4
      RST     M224  ; A D Plates C1
      MPS
      ANI     M224  ; A D Plates C1
      SET     M225  ; A U Plates C1
      MRD
      AND     M225  ; A U Plates C1
      AND     M13  ; SS Cyl U Plates
      RST     M227  ; A D Cyl Rotate_C1ư
      MRD
      ANI     M227  ; A D Cyl Rotate_C1ư
      SET     M226  ; A U Cyl Rotate_C1
      MRD
      AND     M226  ; A U Cyl Rotate_C1
      AND     M15  ; SS U Cyl U Rotate
      RST     M257  ; A Cyl Rotate Add Plate
      ANI     M257  ; A Cyl Rotate Add Plate
      SET     M258  ; A Cyl Rotate Home
      MPP
      AND     M258  ; A Cyl Rotate Home
      AND     M14  ; Home_Cyl_Rotate
      AND     M226  ; A U Cyl Rotate_C1
      AND     M15  ; SS U Cyl U Rotate
      MOV     K0 Add_Plates_C1
; Out Product C1
855   LD      M201  ; En_Auto_C1
      AND=    Out_Product_C1 K0
      RST     M215  ; A FWD Conv RGV
      RST     M211  ; A REV Conv C1
      RST     M216  ; A Rev Conv RGV
      RST     M214  ; AUTO CONVEYOR ROLLER 1
; Safety Out Product
866   LD>=    Out_Product_C1 K3
      OUT     Codition_C2
872   LD      M56  ; SS Home RGV
      ANI     M57  ; SS TF RGV
      RST     M249  ; AU_NÂNG_STOPER_TRC
      SET     M250  ; AU_Hạ_SToper_trước
      RST     M252  ; AU_Hạ_SToper_SAU
      SET     M251  ; AU_Nâng_SToper_SAU
878   LD      M57  ; SS TF RGV
      ANI     M56  ; SS Home RGV
      SET     M221  ; AU_Hạ stoper bell
      RST     M222  ; Nâng stoper bell
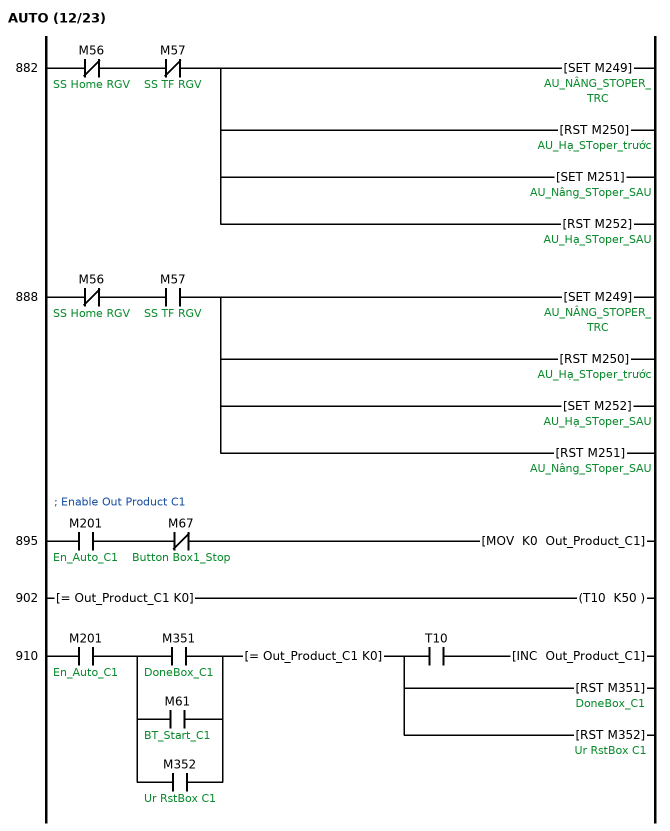
882   LDI     M56  ; SS Home RGV
      ANI     M57  ; SS TF RGV
      SET     M249  ; AU_NÂNG_STOPER_TRC
      RST     M250  ; AU_Hạ_SToper_trước
      SET     M251  ; AU_Nâng_SToper_SAU
      RST     M252  ; AU_Hạ_SToper_SAU
888   LDI     M56  ; SS Home RGV
      AND     M57  ; SS TF RGV
      SET     M249  ; AU_NÂNG_STOPER_TRC
      RST     M250  ; AU_Hạ_SToper_trước
      SET     M252  ; AU_Hạ_SToper_SAU
      RST     M251  ; AU_Nâng_SToper_SAU
; Enable Out Product C1
895   LD      M201  ; En_Auto_C1
      ANI     M67  ; Button Box1_Stop
      MOV     K0 Out_Product_C1
902   LD=     Out_Product_C1 K0
      OUT     T10 K50
910   LD      M201  ; En_Auto_C1
      LD      M351  ; DoneBox_C1
      OR      M61  ; BT_Start_C1
      OR      M352  ; Ur RstBox C1
      ANB
      AND=    Out_Product_C1 K0
      MPS
      AND     T10
      INC     Out_Product_C1
      MPP
      RST     M351  ; DoneBox_C1
      RST     M352  ; Ur RstBox C1
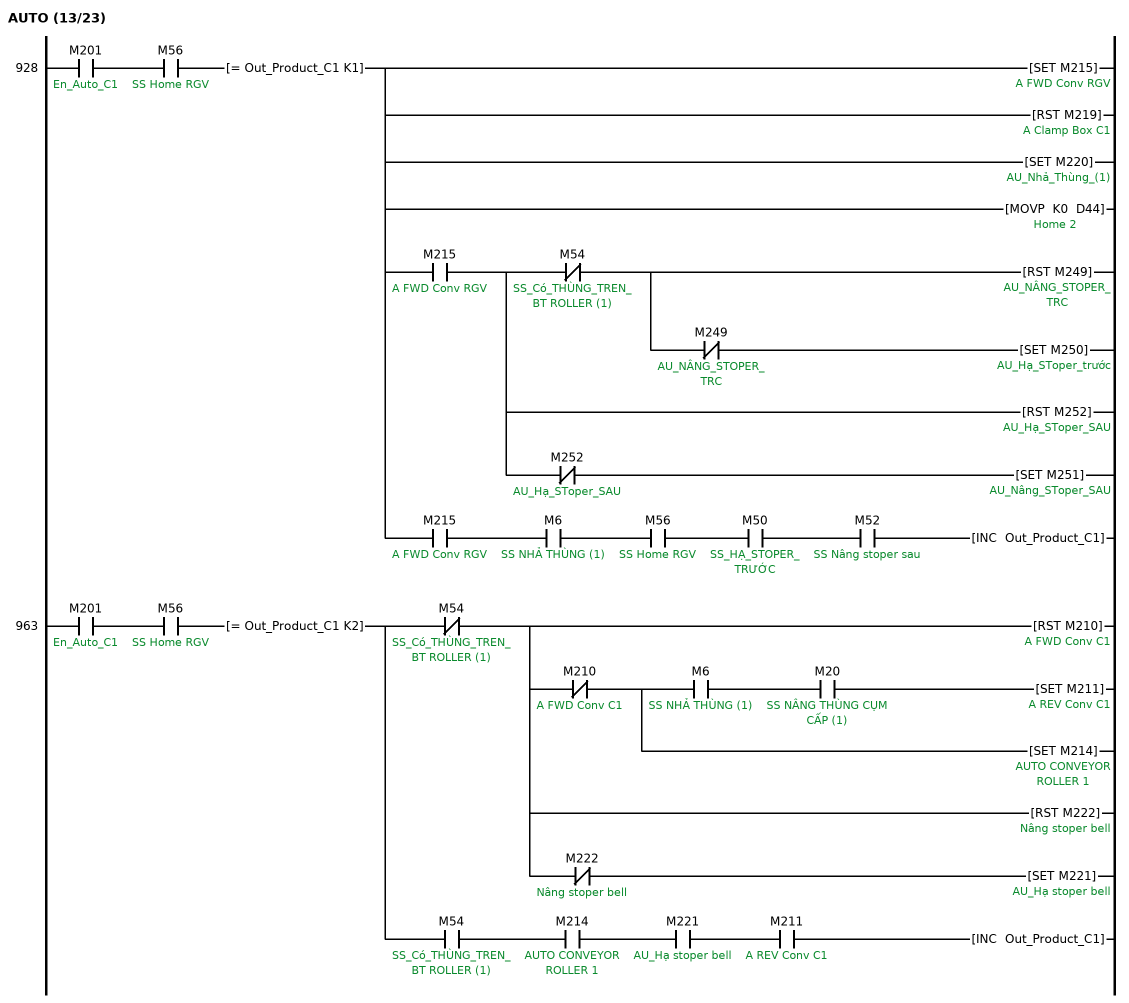
928   LD      M201  ; En_Auto_C1
      AND     M56  ; SS Home RGV
      AND=    Out_Product_C1 K1
      SET     M215  ; A FWD Conv RGV
      RST     M219  ; A Clamp Box C1
      SET     M220  ; AU_Nhả_Thùng_(1)
      MOVP    K0 D44  ; Home 2
      MPS
      AND     M215  ; A FWD Conv RGV
      MPS
      ANI     M54  ; SS_Có_THÙNG_TREN_BT ROLLER (1)
      RST     M249  ; AU_NÂNG_STOPER_TRC
      ANI     M249  ; AU_NÂNG_STOPER_TRC
      SET     M250  ; AU_Hạ_SToper_trước
      MPP
      RST     M252  ; AU_Hạ_SToper_SAU
      ANI     M252  ; AU_Hạ_SToper_SAU
      SET     M251  ; AU_Nâng_SToper_SAU
      MPP
      AND     M215  ; A FWD Conv RGV
      AND     M6  ; SS NHẢ THÙNG (1)
      AND     M56  ; SS Home RGV
      AND     M50  ; SS_HẠ_STOPER_TRƯỚC
      AND     M52  ; SS Nâng stoper sau
      INC     Out_Product_C1
963   LD      M201  ; En_Auto_C1
      AND     M56  ; SS Home RGV
      AND=    Out_Product_C1 K2
      MPS
      ANI     M54  ; SS_Có_THÙNG_TREN_BT ROLLER (1)
      RST     M210  ; A FWD Conv C1
      MPS
      ANI     M210  ; A FWD Conv C1
      MPS
      AND     M6  ; SS NHẢ THÙNG (1)
      AND     M20  ; SS NÂNG THÙNG CỤM CẤP (1)
      SET     M211  ; A REV Conv C1
      MPP
      SET     M214  ; AUTO CONVEYOR ROLLER 1
      MPP
      RST     M222  ; Nâng stoper bell
      ANI     M222  ; Nâng stoper bell
      SET     M221  ; AU_Hạ stoper bell
      MPP
      AND     M54  ; SS_Có_THÙNG_TREN_BT ROLLER (1)
      AND     M214  ; AUTO CONVEYOR ROLLER 1
      AND     M221  ; AU_Hạ stoper bell
      AND     M211  ; A REV Conv C1
      INC     Out_Product_C1
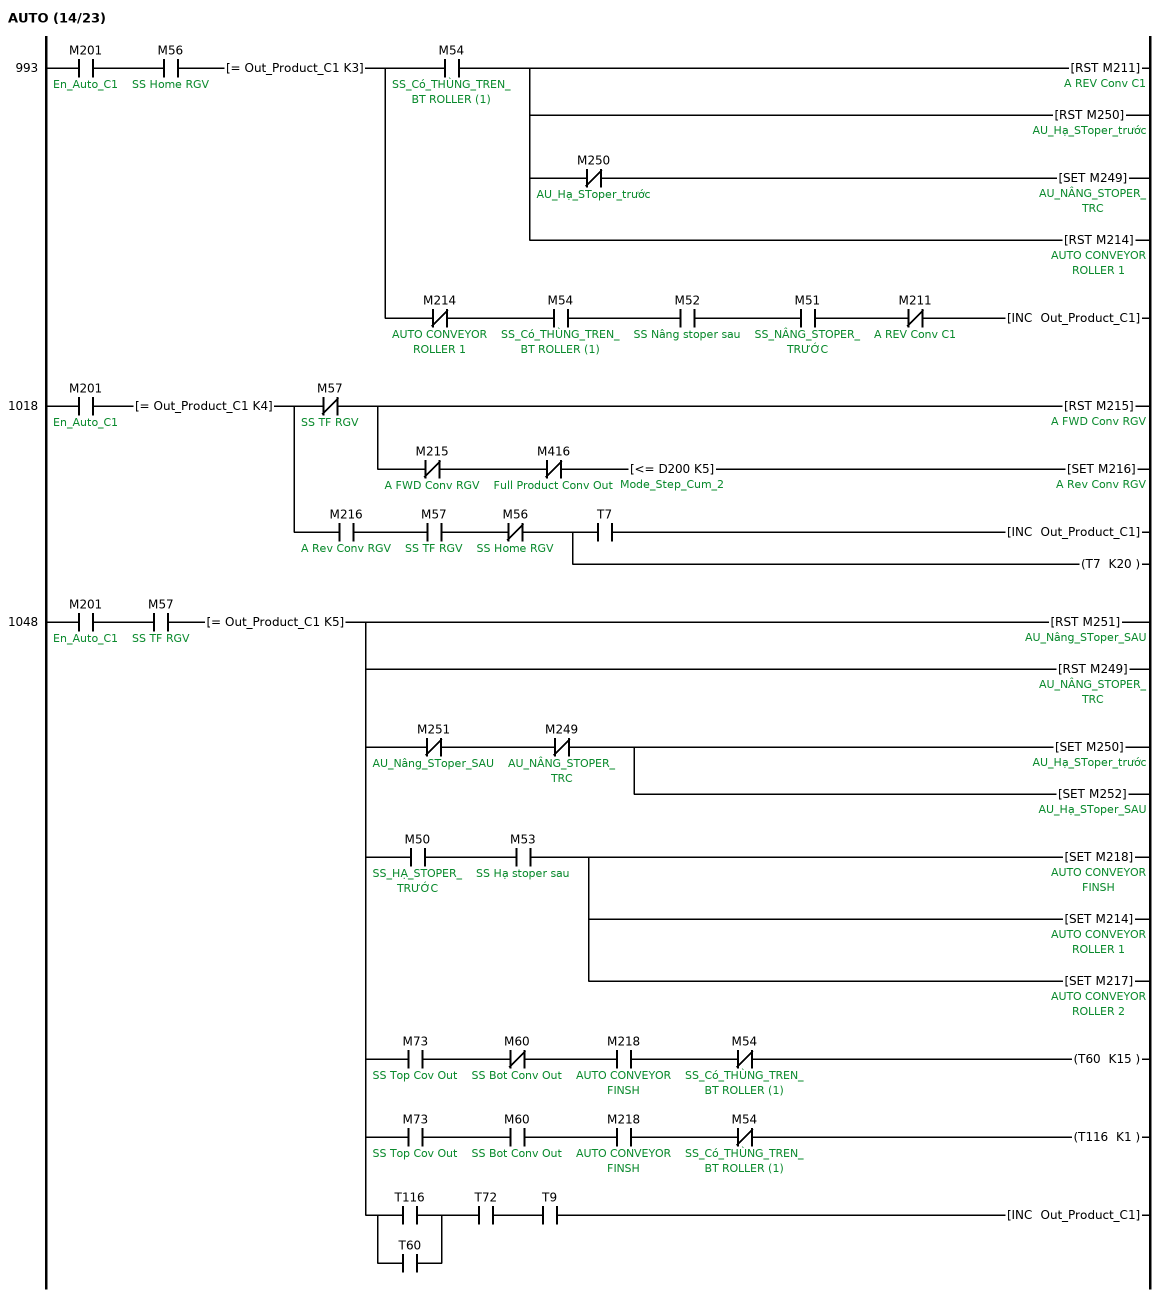
993   LD      M201  ; En_Auto_C1
      AND     M56  ; SS Home RGV
      AND=    Out_Product_C1 K3
      MPS
      AND     M54  ; SS_Có_THÙNG_TREN_BT ROLLER (1)
      RST     M211  ; A REV Conv C1
      RST     M250  ; AU_Hạ_SToper_trước
      MPS
      ANI     M250  ; AU_Hạ_SToper_trước
      SET     M249  ; AU_NÂNG_STOPER_TRC
      MPP
      RST     M214  ; AUTO CONVEYOR ROLLER 1
      MPP
      ANI     M214  ; AUTO CONVEYOR ROLLER 1
      AND     M54  ; SS_Có_THÙNG_TREN_BT ROLLER (1)
      AND     M52  ; SS Nâng stoper sau
      AND     M51  ; SS_NÂNG_STOPER_TRƯỚC
      ANI     M211  ; A REV Conv C1
      INC     Out_Product_C1
1018  LD      M201  ; En_Auto_C1
      AND=    Out_Product_C1 K4
      MPS
      ANI     M57  ; SS TF RGV
      RST     M215  ; A FWD Conv RGV
      ANI     M215  ; A FWD Conv RGV
      ANI     M416  ; Full Product Conv Out
      AND<=   D200 K5  ; Mode_Step_Cum_2
      SET     M216  ; A Rev Conv RGV
      MPP
      AND     M216  ; A Rev Conv RGV
      AND     M57  ; SS TF RGV
      ANI     M56  ; SS Home RGV
      MPS
      AND     T7
      INC     Out_Product_C1
      MPP
      OUT     T7 K20
1048  LD      M201  ; En_Auto_C1
      AND     M57  ; SS TF RGV
      AND=    Out_Product_C1 K5
      RST     M251  ; AU_Nâng_SToper_SAU
      RST     M249  ; AU_NÂNG_STOPER_TRC
      MPS
      ANI     M251  ; AU_Nâng_SToper_SAU
      ANI     M249  ; AU_NÂNG_STOPER_TRC
      SET     M250  ; AU_Hạ_SToper_trước
      SET     M252  ; AU_Hạ_SToper_SAU
      MRD
      AND     M50  ; SS_HẠ_STOPER_TRƯỚC
      AND     M53  ; SS Hạ stoper sau
      SET     M218  ; AUTO CONVEYOR FINSH
      SET     M214  ; AUTO CONVEYOR ROLLER 1
      SET     M217  ; AUTO CONVEYOR ROLLER 2
      MRD
      AND     M73  ; SS Top Cov Out
      ANI     M60  ; SS Bot Conv Out
      AND     M218  ; AUTO CONVEYOR FINSH
      ANI     M54  ; SS_Có_THÙNG_TREN_BT ROLLER (1)
      OUT     T60 K15
      MRD
      AND     M73  ; SS Top Cov Out
      AND     M60  ; SS Bot Conv Out
      AND     M218  ; AUTO CONVEYOR FINSH
      ANI     M54  ; SS_Có_THÙNG_TREN_BT ROLLER (1)
      OUT     T116 K1
      MPP
      LD      T116
      OR      T60
      ANB
      AND     T72
      AND     T9
      INC     Out_Product_C1
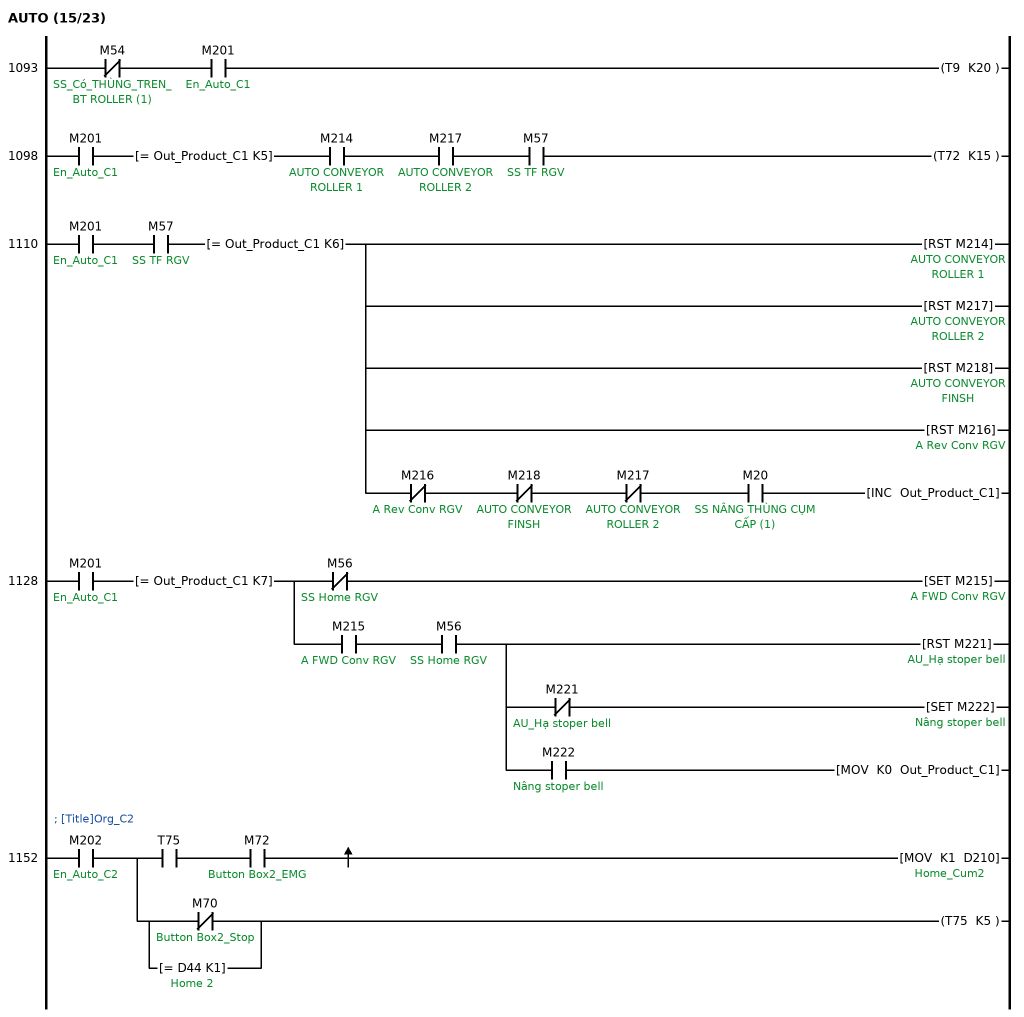
1093  LDI     M54  ; SS_Có_THÙNG_TREN_BT ROLLER (1)
      AND     M201  ; En_Auto_C1
      OUT     T9 K20
1098  LD      M201  ; En_Auto_C1
      AND=    Out_Product_C1 K5
      AND     M214  ; AUTO CONVEYOR ROLLER 1
      AND     M217  ; AUTO CONVEYOR ROLLER 2
      AND     M57  ; SS TF RGV
      OUT     T72 K15
1110  LD      M201  ; En_Auto_C1
      AND     M57  ; SS TF RGV
      AND=    Out_Product_C1 K6
      RST     M214  ; AUTO CONVEYOR ROLLER 1
      RST     M217  ; AUTO CONVEYOR ROLLER 2
      RST     M218  ; AUTO CONVEYOR FINSH
      RST     M216  ; A Rev Conv RGV
      ANI     M216  ; A Rev Conv RGV
      ANI     M218  ; AUTO CONVEYOR FINSH
      ANI     M217  ; AUTO CONVEYOR ROLLER 2
      AND     M20  ; SS NÂNG THÙNG CỤM CẤP (1)
      INC     Out_Product_C1
1128  LD      M201  ; En_Auto_C1
      AND=    Out_Product_C1 K7
      MPS
      ANI     M56  ; SS Home RGV
      SET     M215  ; A FWD Conv RGV
      MPP
      AND     M215  ; A FWD Conv RGV
      AND     M56  ; SS Home RGV
      RST     M221  ; AU_Hạ stoper bell
      MPS
      ANI     M221  ; AU_Hạ stoper bell
      SET     M222  ; Nâng stoper bell
      MPP
      AND     M222  ; Nâng stoper bell
      MOV     K0 Out_Product_C1
; [Title]Org_C2
1152  LD      M202  ; En_Auto_C2
      MPS
      AND     T75
      AND     M72  ; Button Box2_EMG
      MEP
      MOV     K1 D210  ; Home_Cum2
      MPP
      LDI     M70  ; Button Box2_Stop
      OR=     D44 K1  ; Home 2
      ANB
      OUT     T75 K5
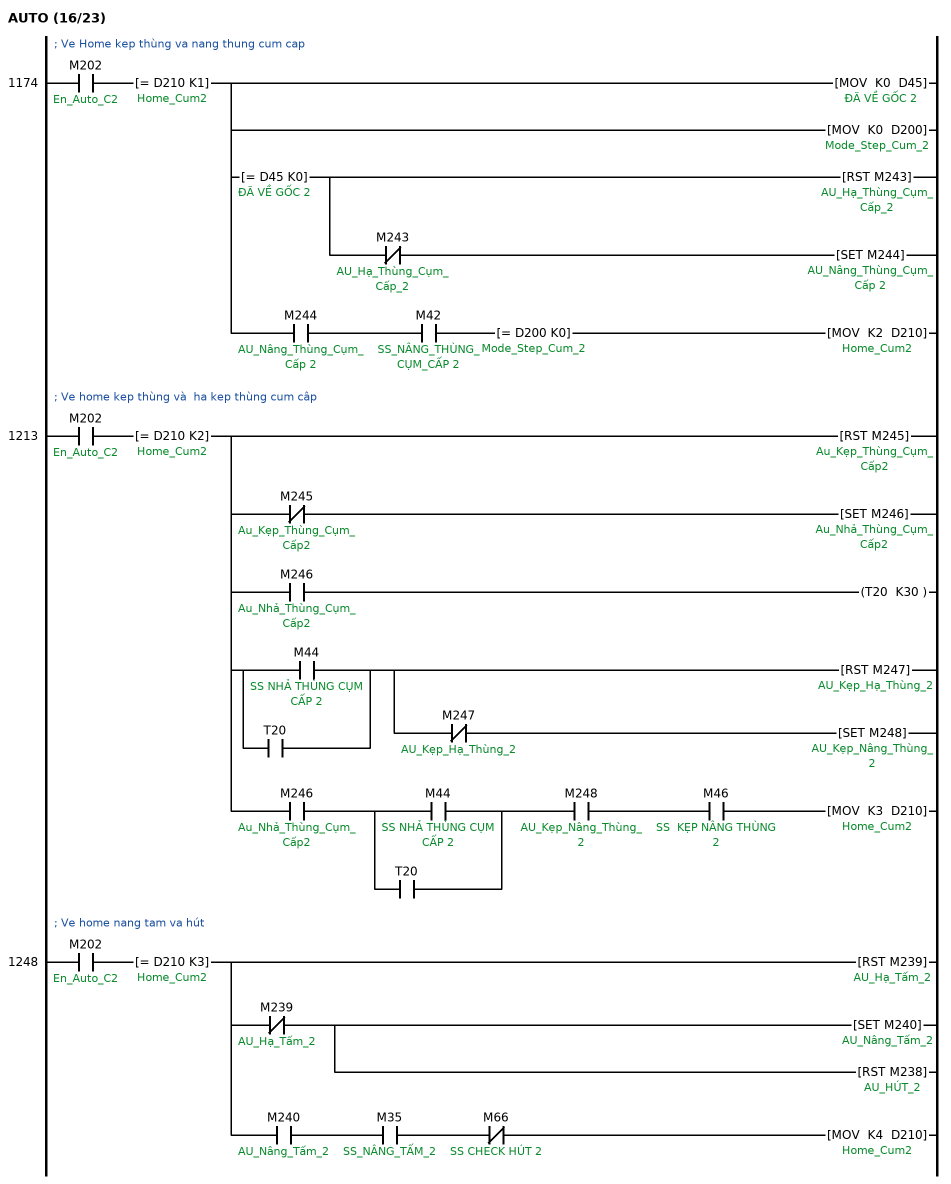
; Ve Home kep thùng va nang thung cum cap
1174  LD      M202  ; En_Auto_C2
      AND=    D210 K1  ; Home_Cum2
      MOV     K0 D45  ; ĐÃ VỀ GỐC 2
      MOV     K0 D200
      MPS
      AND=    D45 K0  ; ĐÃ VỀ GỐC 2
      RST     M243  ; AU_Hạ_Thùng_Cụm_Cấp_2
      ANI     M243  ; AU_Hạ_Thùng_Cụm_Cấp_2
      SET     M244  ; AU_Nâng_Thùng_Cụm_Cấp 2
      MPP
      AND     M244  ; AU_Nâng_Thùng_Cụm_Cấp 2
      AND     M42  ; SS_NÂNG_THÙNG_CỤM_CẤP 2
      AND=    D200 K0  ; Mode_Step_Cum_2
      MOV     K2 D210
; Ve home kep thùng và  ha kep thùng cum câp
1213  LD      M202  ; En_Auto_C2
      AND=    D210 K2  ; Home_Cum2
      RST     M245  ; Au_Kẹp_Thùng_Cụm_Cấp2
      MPS
      ANI     M245  ; Au_Kẹp_Thùng_Cụm_Cấp2
      SET     M246  ; Au_Nhả_Thùng_Cụm_Cấp2
      MRD
      AND     M246  ; Au_Nhả_Thùng_Cụm_Cấp2
      OUT     T20 K30
      MRD
      LD      M44  ; SS NHẢ THÙNG CỤM CẤP 2
      OR      T20
      ANB
      RST     M247  ; AU_Kẹp_Hạ_Thùng_2
      ANI     M247  ; AU_Kẹp_Hạ_Thùng_2
      SET     M248  ; AU_Kẹp_Nâng_Thùng_2
      MPP
      AND     M246  ; Au_Nhả_Thùng_Cụm_Cấp2
      LD      M44  ; SS NHẢ THÙNG CỤM CẤP 2
      OR      T20
      ANB
      AND     M248  ; AU_Kẹp_Nâng_Thùng_2
      AND     M46  ; SS  KẸP NÂNG THÙNG 2
      MOV     K3 D210
; Ve home nang tam va hút
1248  LD      M202  ; En_Auto_C2
      AND=    D210 K3  ; Home_Cum2
      RST     M239  ; AU_Hạ_Tấm_2
      MPS
      ANI     M239  ; AU_Hạ_Tấm_2
      SET     M240  ; AU_Nâng_Tấm_2
      RST     M238  ; AU_HÚT_2
      MPP
      AND     M240  ; AU_Nâng_Tấm_2
      AND     M35  ; SS_NÂNG_TẤM_2
      ANI     M66  ; SS CHECK HÚT 2
      MOV     K4 D210
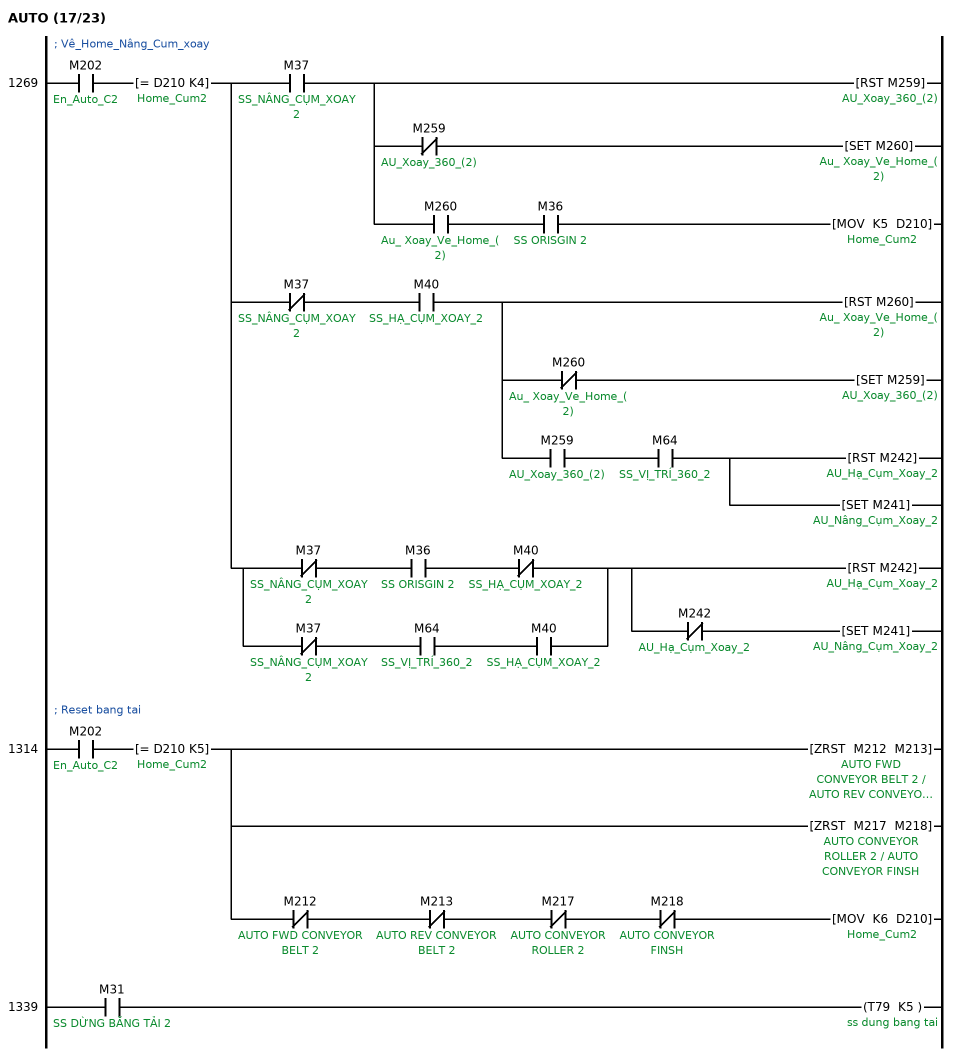
; Vê_Home_Nâng_Cum_xoay
1269  LD      M202  ; En_Auto_C2
      AND=    D210 K4  ; Home_Cum2
      MPS
      AND     M37  ; SS_NÂNG_CỤM_XOAY 2
      RST     M259  ; AU_Xoay_360_(2)
      MPS
      ANI     M259  ; AU_Xoay_360_(2)
      SET     M260  ; Au_ Xoay_Ve_Home_(2)
      MPP
      AND     M260  ; Au_ Xoay_Ve_Home_(2)
      AND     M36  ; SS ORISGIN 2
      MOV     K5 D210
      MRD
      ANI     M37  ; SS_NÂNG_CỤM_XOAY 2
      AND     M40  ; SS_HẠ_CỤM_XOAY_2
      RST     M260  ; Au_ Xoay_Ve_Home_(2)
      MPS
      ANI     M260  ; Au_ Xoay_Ve_Home_(2)
      SET     M259  ; AU_Xoay_360_(2)
      MPP
      AND     M259  ; AU_Xoay_360_(2)
      AND     M64  ; SS_VỊ_TRÍ_360_2
      RST     M242  ; AU_Hạ_Cụm_Xoay_2
      SET     M241  ; AU_Nâng_Cụm_Xoay_2
      MPP
      LDI     M37  ; SS_NÂNG_CỤM_XOAY 2
      AND     M36  ; SS ORISGIN 2
      ANI     M40  ; SS_HẠ_CỤM_XOAY_2
      LDI     M37  ; SS_NÂNG_CỤM_XOAY 2
      AND     M64  ; SS_VỊ_TRÍ_360_2
      AND     M40  ; SS_HẠ_CỤM_XOAY_2
      ORB
      ANB
      RST     M242  ; AU_Hạ_Cụm_Xoay_2
      ANI     M242  ; AU_Hạ_Cụm_Xoay_2
      SET     M241  ; AU_Nâng_Cụm_Xoay_2
; Reset bang tai
1314  LD      M202  ; En_Auto_C2
      AND=    D210 K5  ; Home_Cum2
      ZRST    M212 M213  ; AUTO FWD CONVEYOR BELT 2 / AUTO REV CONVEYOR BELT 2
      ZRST    M217 M218
      ANI     M212  ; AUTO FWD CONVEYOR BELT 2
      ANI     M213  ; AUTO REV CONVEYOR BELT 2
      ANI     M217  ; AUTO CONVEYOR ROLLER 2
      ANI     M218  ; AUTO CONVEYOR FINSH
      MOV     K6 D210
1339  LD      M31  ; SS DỪNG BĂNG TẢI 2
      OUT     T79 K5  ; ss dung bang tai
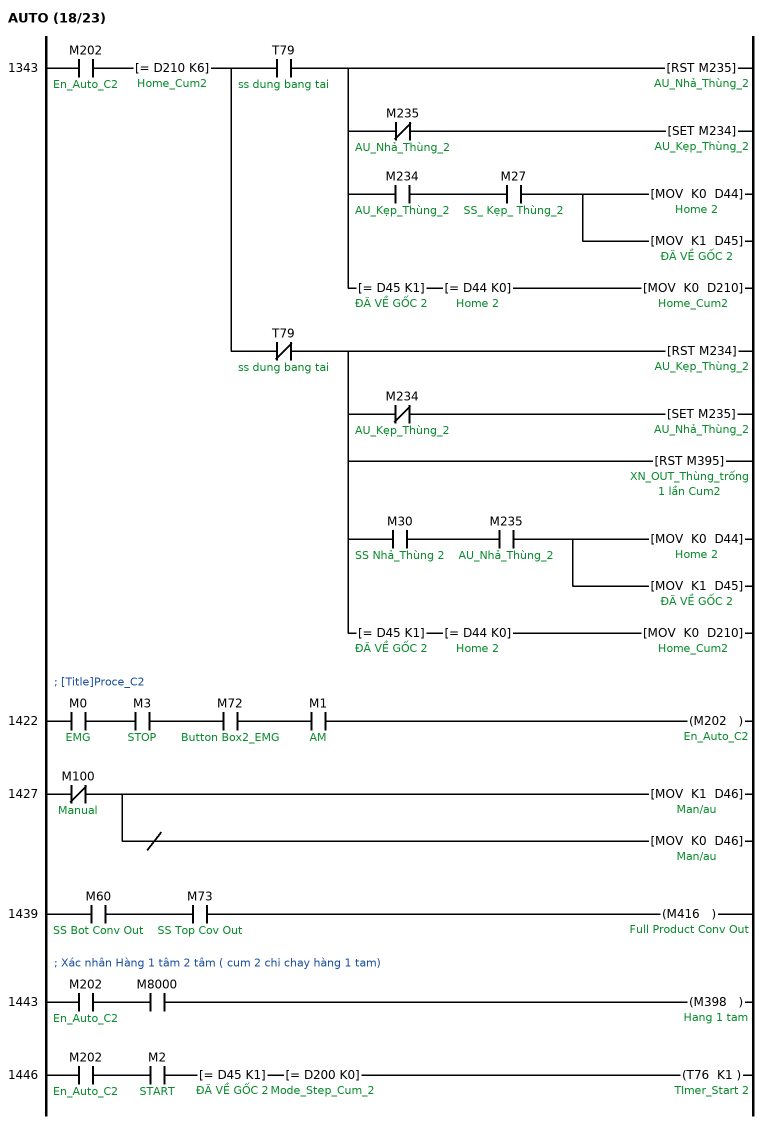
1343  LD      M202  ; En_Auto_C2
      AND=    D210 K6  ; Home_Cum2
      MPS
      AND     T79  ; ss dung bang tai
      RST     M235  ; AU_Nhả_Thùng_2
      MPS
      ANI     M235  ; AU_Nhả_Thùng_2
      SET     M234  ; AU_Kẹp_Thùng_2
      MRD
      AND     M234  ; AU_Kẹp_Thùng_2
      AND     M27  ; SS_ Kẹp_ Thùng_2
      MOV     K0 D44
      MOV     K1 D45
      MPP
      AND=    D45 K1  ; ĐÃ VỀ GỐC 2
      AND=    D44 K0  ; Home 2
      MOV     K0 D210
      MPP
      ANI     T79  ; ss dung bang tai
      RST     M234  ; AU_Kẹp_Thùng_2
      MPS
      ANI     M234  ; AU_Kẹp_Thùng_2
      SET     M235  ; AU_Nhả_Thùng_2
      MPP
      RST     M395  ; XN_OUT_Thùng_trống 1 lần Cum2
      MPS
      AND     M30  ; SS Nhả_Thùng 2
      AND     M235  ; AU_Nhả_Thùng_2
      MOV     K0 D44
      MOV     K1 D45
      MPP
      AND=    D45 K1  ; ĐÃ VỀ GỐC 2
      AND=    D44 K0  ; Home 2
      MOV     K0 D210
; [Title]Proce_C2
1422  LD      M0  ; EMG
      AND     M3  ; STOP
      AND     M72  ; Button Box2_EMG
      AND     M1  ; AM
      OUT     M202  ; En_Auto_C2
1427  LDI     M100  ; Manual
      MOV     K1 D46  ; Man/au
      INV
      MOV     K0 D46
1439  LD      M60  ; SS Bot Conv Out
      AND     M73  ; SS Top Cov Out
      OUT     M416  ; Full Product Conv Out
; Xác nhân Hàng 1 tâm 2 tâm ( cum 2 chi chay hàng 1 tam)
1443  LD      M202  ; En_Auto_C2
      AND     M8000
      OUT     M398  ; Hang 1 tam
1446  LD      M202  ; En_Auto_C2
      AND     M2  ; START
      AND=    D45 K1  ; ĐÃ VỀ GỐC 2
      AND=    D200 K0  ; Mode_Step_Cum_2
      OUT     T76 K1  ; TImer_Start 2
